*)
END_ACTION
ACTION derevo_write:
_CFC_ (* Continuous Function Chart, elements in execution order *)
_END_CFC_
END_ACTION
ACTION eibPort_climate:
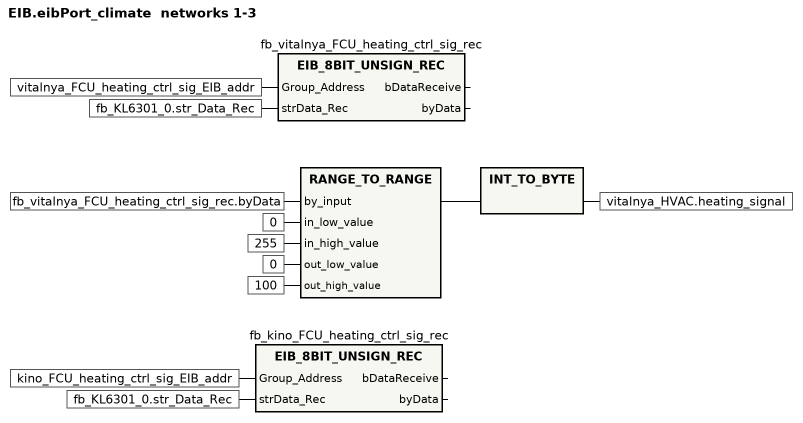
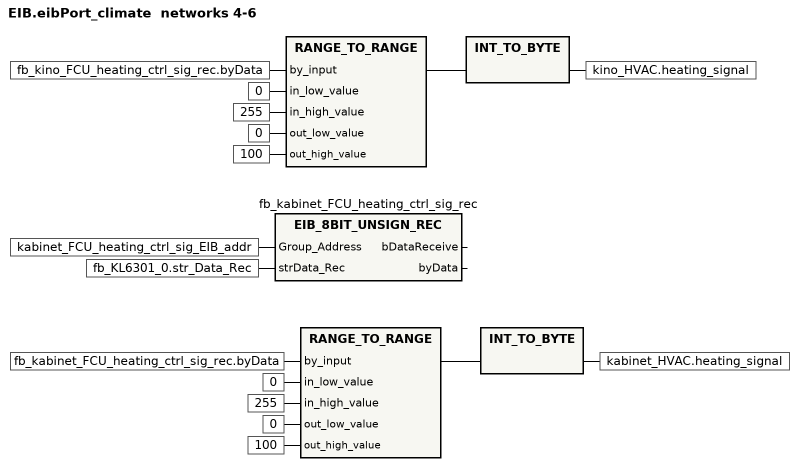
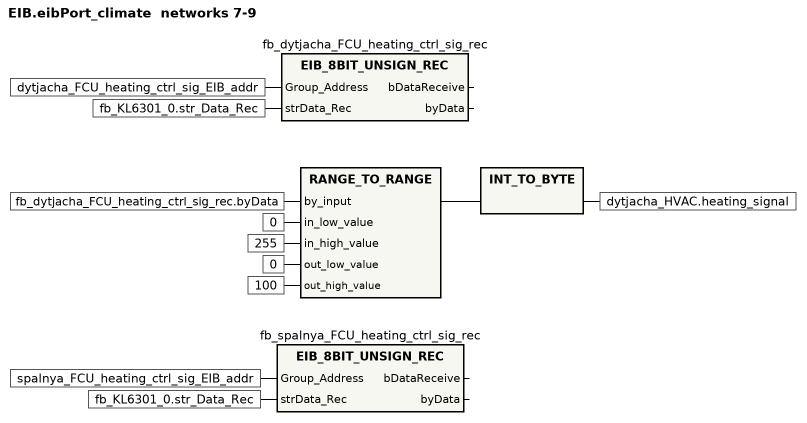
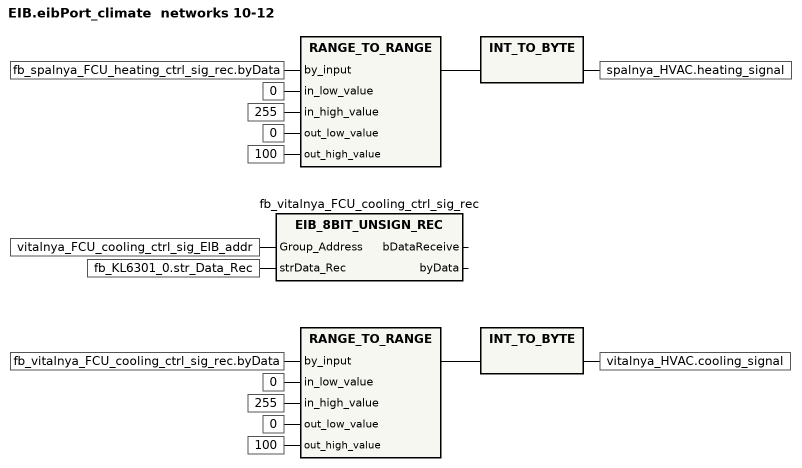
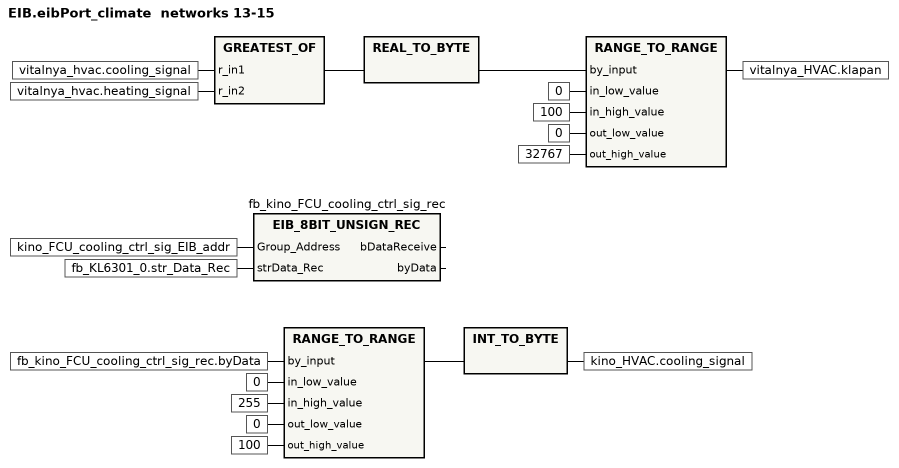
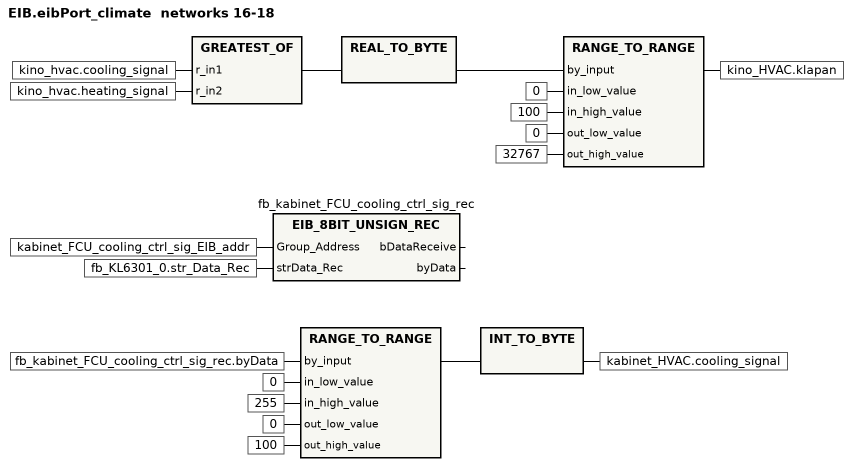
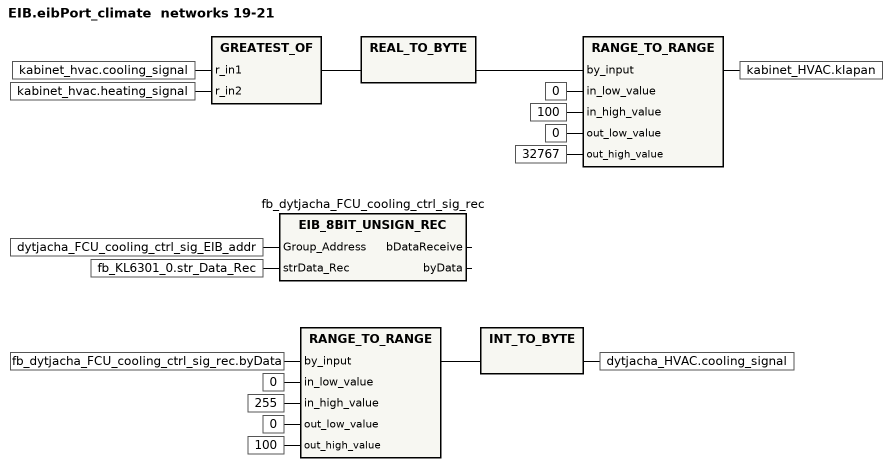
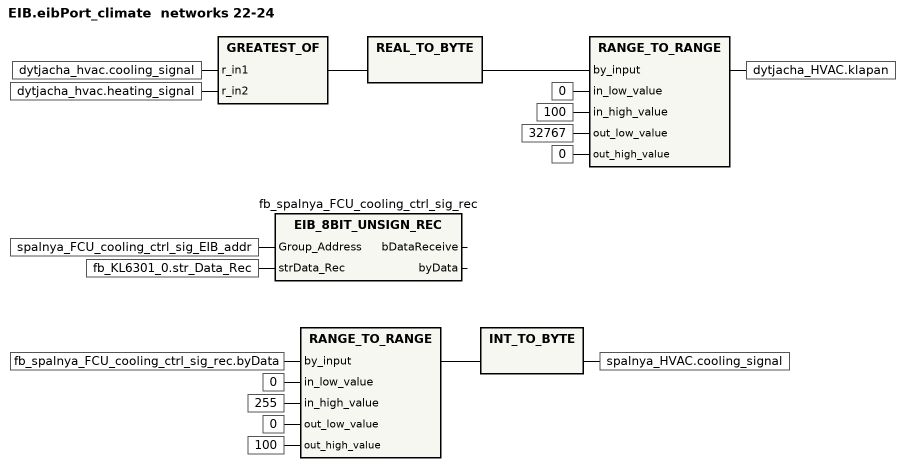
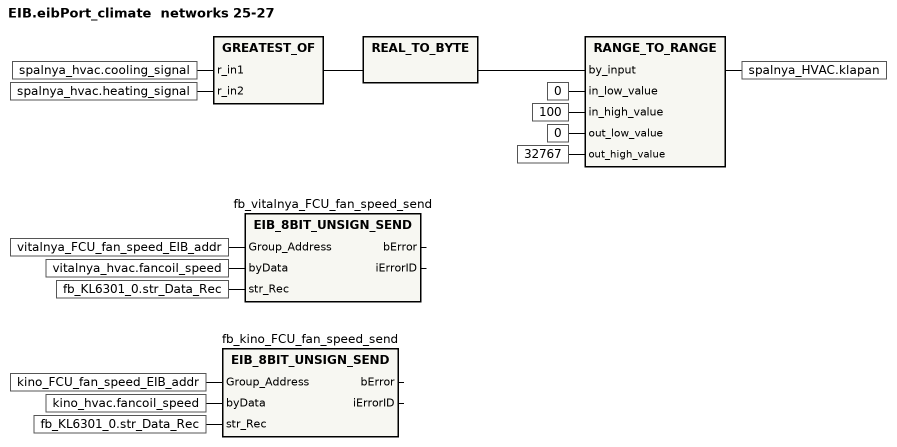
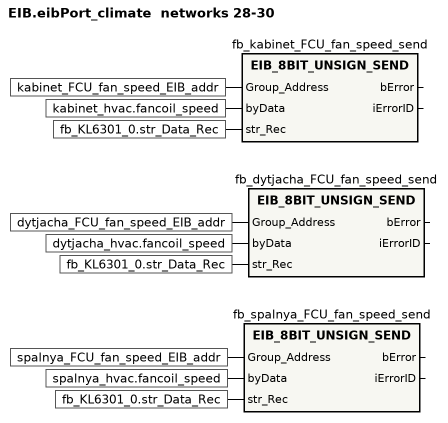
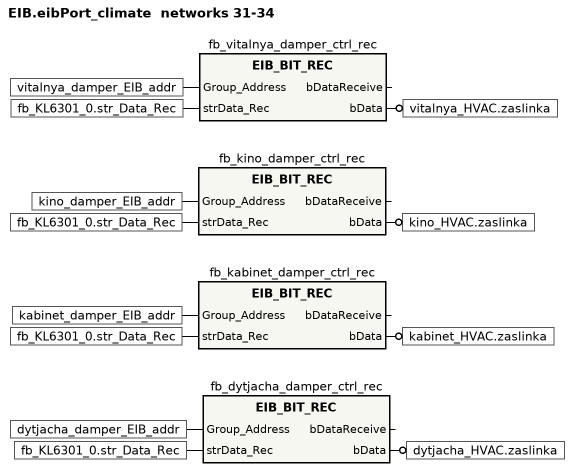
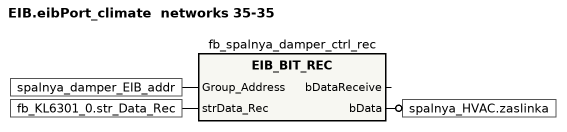
_FBD_ (* Function Block Diagram *)
NETWORK 1
	fb_vitalnya_FCU_heating_ctrl_sig_rec:EIB_8BIT_UNSIGN_REC(Group_Address: vitalnya_FCU_heating_ctrl_sig_EIB_addr, strData_Rec: fb_KL6301_0.str_Data_Rec)
NETWORK 2
	INT_TO_BYTE(RANGE_TO_RANGE(by_input: fb_vitalnya_FCU_heating_ctrl_sig_rec.byData, in_low_value: 0, in_high_value: 255, out_low_value: 0, out_high_value: 100)) => vitalnya_HVAC.heating_signal
NETWORK 3
	fb_kino_FCU_heating_ctrl_sig_rec:EIB_8BIT_UNSIGN_REC(Group_Address: kino_FCU_heating_ctrl_sig_EIB_addr, strData_Rec: fb_KL6301_0.str_Data_Rec)
NETWORK 4
	INT_TO_BYTE(RANGE_TO_RANGE(by_input: fb_kino_FCU_heating_ctrl_sig_rec.byData, in_low_value: 0, in_high_value: 255, out_low_value: 0, out_high_value: 100)) => kino_HVAC.heating_signal
NETWORK 5
	fb_kabinet_FCU_heating_ctrl_sig_rec:EIB_8BIT_UNSIGN_REC(Group_Address: kabinet_FCU_heating_ctrl_sig_EIB_addr, strData_Rec: fb_KL6301_0.str_Data_Rec)
NETWORK 6
	INT_TO_BYTE(RANGE_TO_RANGE(by_input: fb_kabinet_FCU_heating_ctrl_sig_rec.byData, in_low_value: 0, in_high_value: 255, out_low_value: 0, out_high_value: 100)) => kabinet_HVAC.heating_signal
NETWORK 7
	fb_dytjacha_FCU_heating_ctrl_sig_rec:EIB_8BIT_UNSIGN_REC(Group_Address: dytjacha_FCU_heating_ctrl_sig_EIB_addr, strData_Rec: fb_KL6301_0.str_Data_Rec)
NETWORK 8
	INT_TO_BYTE(RANGE_TO_RANGE(by_input: fb_dytjacha_FCU_heating_ctrl_sig_rec.byData, in_low_value: 0, in_high_value: 255, out_low_value: 0, out_high_value: 100)) => dytjacha_HVAC.heating_signal
NETWORK 9
	fb_spalnya_FCU_heating_ctrl_sig_rec:EIB_8BIT_UNSIGN_REC(Group_Address: spalnya_FCU_heating_ctrl_sig_EIB_addr, strData_Rec: fb_KL6301_0.str_Data_Rec)
NETWORK 10
	INT_TO_BYTE(RANGE_TO_RANGE(by_input: fb_spalnya_FCU_heating_ctrl_sig_rec.byData, in_low_value: 0, in_high_value: 255, out_low_value: 0, out_high_value: 100)) => spalnya_HVAC.heating_signal
NETWORK 11
	fb_vitalnya_FCU_cooling_ctrl_sig_rec:EIB_8BIT_UNSIGN_REC(Group_Address: vitalnya_FCU_cooling_ctrl_sig_EIB_addr, strData_Rec: fb_KL6301_0.str_Data_Rec)
NETWORK 12
	INT_TO_BYTE(RANGE_TO_RANGE(by_input: fb_vitalnya_FCU_cooling_ctrl_sig_rec.byData, in_low_value: 0, in_high_value: 255, out_low_value: 0, out_high_value: 100)) => vitalnya_HVAC.cooling_signal
NETWORK 13
	RANGE_TO_RANGE(by_input: REAL_TO_BYTE(GREATEST_OF(r_in1: vitalnya_hvac.cooling_signal, r_in2: vitalnya_hvac.heating_signal)), in_low_value: 0, in_high_value: 100, out_low_value: 0, out_high_value: 32767) => vitalnya_HVAC.klapan
NETWORK 14
	fb_kino_FCU_cooling_ctrl_sig_rec:EIB_8BIT_UNSIGN_REC(Group_Address: kino_FCU_cooling_ctrl_sig_EIB_addr, strData_Rec: fb_KL6301_0.str_Data_Rec)
NETWORK 15
	INT_TO_BYTE(RANGE_TO_RANGE(by_input: fb_kino_FCU_cooling_ctrl_sig_rec.byData, in_low_value: 0, in_high_value: 255, out_low_value: 0, out_high_value: 100)) => kino_HVAC.cooling_signal
NETWORK 16
	RANGE_TO_RANGE(by_input: REAL_TO_BYTE(GREATEST_OF(r_in1: kino_hvac.cooling_signal, r_in2: kino_hvac.heating_signal)), in_low_value: 0, in_high_value: 100, out_low_value: 0, out_high_value: 32767) => kino_HVAC.klapan
NETWORK 17
	fb_kabinet_FCU_cooling_ctrl_sig_rec:EIB_8BIT_UNSIGN_REC(Group_Address: kabinet_FCU_cooling_ctrl_sig_EIB_addr, strData_Rec: fb_KL6301_0.str_Data_Rec)
NETWORK 18
	INT_TO_BYTE(RANGE_TO_RANGE(by_input: fb_kabinet_FCU_cooling_ctrl_sig_rec.byData, in_low_value: 0, in_high_value: 255, out_low_value: 0, out_high_value: 100)) => kabinet_HVAC.cooling_signal
NETWORK 19
	RANGE_TO_RANGE(by_input: REAL_TO_BYTE(GREATEST_OF(r_in1: kabinet_hvac.cooling_signal, r_in2: kabinet_hvac.heating_signal)), in_low_value: 0, in_high_value: 100, out_low_value: 0, out_high_value: 32767) => kabinet_HVAC.klapan
NETWORK 20
	fb_dytjacha_FCU_cooling_ctrl_sig_rec:EIB_8BIT_UNSIGN_REC(Group_Address: dytjacha_FCU_cooling_ctrl_sig_EIB_addr, strData_Rec: fb_KL6301_0.str_Data_Rec)
NETWORK 21
	INT_TO_BYTE(RANGE_TO_RANGE(by_input: fb_dytjacha_FCU_cooling_ctrl_sig_rec.byData, in_low_value: 0, in_high_value: 255, out_low_value: 0, out_high_value: 100)) => dytjacha_HVAC.cooling_signal
NETWORK 22
	RANGE_TO_RANGE(by_input: REAL_TO_BYTE(GREATEST_OF(r_in1: dytjacha_hvac.cooling_signal, r_in2: dytjacha_hvac.heating_signal)), in_low_value: 0, in_high_value: 100, out_low_value: 32767, out_high_value: 0) => dytjacha_HVAC.klapan
NETWORK 23
	fb_spalnya_FCU_cooling_ctrl_sig_rec:EIB_8BIT_UNSIGN_REC(Group_Address: spalnya_FCU_cooling_ctrl_sig_EIB_addr, strData_Rec: fb_KL6301_0.str_Data_Rec)
NETWORK 24
	INT_TO_BYTE(RANGE_TO_RANGE(by_input: fb_spalnya_FCU_cooling_ctrl_sig_rec.byData, in_low_value: 0, in_high_value: 255, out_low_value: 0, out_high_value: 100)) => spalnya_HVAC.cooling_signal
NETWORK 25
	RANGE_TO_RANGE(by_input: REAL_TO_BYTE(GREATEST_OF(r_in1: spalnya_hvac.cooling_signal, r_in2: spalnya_hvac.heating_signal)), in_low_value: 0, in_high_value: 100, out_low_value: 0, out_high_value: 32767) => spalnya_HVAC.klapan
NETWORK 26
	fb_vitalnya_FCU_fan_speed_send:EIB_8BIT_UNSIGN_SEND(Group_Address: vitalnya_FCU_fan_speed_EIB_addr, byData: vitalnya_hvac.fancoil_speed, str_Rec: fb_KL6301_0.str_Data_Rec)
NETWORK 27
	fb_kino_FCU_fan_speed_send:EIB_8BIT_UNSIGN_SEND(Group_Address: kino_FCU_fan_speed_EIB_addr, byData: kino_hvac.fancoil_speed, str_Rec: fb_KL6301_0.str_Data_Rec)
NETWORK 28
	fb_kabinet_FCU_fan_speed_send:EIB_8BIT_UNSIGN_SEND(Group_Address: kabinet_FCU_fan_speed_EIB_addr, byData: kabinet_hvac.fancoil_speed, str_Rec: fb_KL6301_0.str_Data_Rec)
NETWORK 29
	fb_dytjacha_FCU_fan_speed_send:EIB_8BIT_UNSIGN_SEND(Group_Address: dytjacha_FCU_fan_speed_EIB_addr, byData: dytjacha_hvac.fancoil_speed, str_Rec: fb_KL6301_0.str_Data_Rec)
NETWORK 30
	fb_spalnya_FCU_fan_speed_send:EIB_8BIT_UNSIGN_SEND(Group_Address: spalnya_FCU_fan_speed_EIB_addr, byData: spalnya_hvac.fancoil_speed, str_Rec: fb_KL6301_0.str_Data_Rec)
NETWORK 31
	fb_vitalnya_damper_ctrl_rec:EIB_BIT_REC(Group_Address: vitalnya_damper_EIB_addr, strData_Rec: fb_KL6301_0.str_Data_Rec, bData => NOT vitalnya_HVAC.zaslinka)
NETWORK 32
	fb_kino_damper_ctrl_rec:EIB_BIT_REC(Group_Address: kino_damper_EIB_addr, strData_Rec: fb_KL6301_0.str_Data_Rec, bData => NOT kino_HVAC.zaslinka)
NETWORK 33
	fb_kabinet_damper_ctrl_rec:EIB_BIT_REC(Group_Address: kabinet_damper_EIB_addr, strData_Rec: fb_KL6301_0.str_Data_Rec, bData => NOT kabinet_HVAC.zaslinka)
NETWORK 34
	fb_dytjacha_damper_ctrl_rec:EIB_BIT_REC(Group_Address: dytjacha_damper_EIB_addr, strData_Rec: fb_KL6301_0.str_Data_Rec, bData => NOT dytjacha_HVAC.zaslinka)
NETWORK 35
	fb_spalnya_damper_ctrl_rec:EIB_BIT_REC(Group_Address: spalnya_damper_EIB_addr, strData_Rec: fb_KL6301_0.str_Data_Rec, bData => NOT spalnya_HVAC.zaslinka)
_END_FBD_
(* the same logic as Structured Text *)
(* Network 1 *)
fb_vitalnya_FCU_heating_ctrl_sig_rec(Group_Address := vitalnya_FCU_heating_ctrl_sig_EIB_addr, strData_Rec := fb_KL6301_0.str_Data_Rec);
(* Network 2 *)
vitalnya_HVAC.heating_signal := INT_TO_BYTE(RANGE_TO_RANGE(by_input := fb_vitalnya_FCU_heating_ctrl_sig_rec.byData, in_low_value := 0, in_high_value := 255, out_low_value := 0, out_high_value := 100));
(* Network 3 *)
fb_kino_FCU_heating_ctrl_sig_rec(Group_Address := kino_FCU_heating_ctrl_sig_EIB_addr, strData_Rec := fb_KL6301_0.str_Data_Rec);
(* Network 4 *)
kino_HVAC.heating_signal := INT_TO_BYTE(RANGE_TO_RANGE(by_input := fb_kino_FCU_heating_ctrl_sig_rec.byData, in_low_value := 0, in_high_value := 255, out_low_value := 0, out_high_value := 100));
(* Network 5 *)
fb_kabinet_FCU_heating_ctrl_sig_rec(Group_Address := kabinet_FCU_heating_ctrl_sig_EIB_addr, strData_Rec := fb_KL6301_0.str_Data_Rec);
(* Network 6 *)
kabinet_HVAC.heating_signal := INT_TO_BYTE(RANGE_TO_RANGE(by_input := fb_kabinet_FCU_heating_ctrl_sig_rec.byData, in_low_value := 0, in_high_value := 255, out_low_value := 0, out_high_value := 100));
(* Network 7 *)
fb_dytjacha_FCU_heating_ctrl_sig_rec(Group_Address := dytjacha_FCU_heating_ctrl_sig_EIB_addr, strData_Rec := fb_KL6301_0.str_Data_Rec);
(* Network 8 *)
dytjacha_HVAC.heating_signal := INT_TO_BYTE(RANGE_TO_RANGE(by_input := fb_dytjacha_FCU_heating_ctrl_sig_rec.byData, in_low_value := 0, in_high_value := 255, out_low_value := 0, out_high_value := 100));
(* Network 9 *)
fb_spalnya_FCU_heating_ctrl_sig_rec(Group_Address := spalnya_FCU_heating_ctrl_sig_EIB_addr, strData_Rec := fb_KL6301_0.str_Data_Rec);
(* Network 10 *)
spalnya_HVAC.heating_signal := INT_TO_BYTE(RANGE_TO_RANGE(by_input := fb_spalnya_FCU_heating_ctrl_sig_rec.byData, in_low_value := 0, in_high_value := 255, out_low_value := 0, out_high_value := 100));
(* Network 11 *)
fb_vitalnya_FCU_cooling_ctrl_sig_rec(Group_Address := vitalnya_FCU_cooling_ctrl_sig_EIB_addr, strData_Rec := fb_KL6301_0.str_Data_Rec);
(* Network 12 *)
vitalnya_HVAC.cooling_signal := INT_TO_BYTE(RANGE_TO_RANGE(by_input := fb_vitalnya_FCU_cooling_ctrl_sig_rec.byData, in_low_value := 0, in_high_value := 255, out_low_value := 0, out_high_value := 100));
(* Network 13 *)
vitalnya_HVAC.klapan := RANGE_TO_RANGE(by_input := REAL_TO_BYTE(GREATEST_OF(r_in1 := vitalnya_hvac.cooling_signal, r_in2 := vitalnya_hvac.heating_signal)), in_low_value := 0, in_high_value := 100, out_low_value := 0, out_high_value := 32767);
(* Network 14 *)
fb_kino_FCU_cooling_ctrl_sig_rec(Group_Address := kino_FCU_cooling_ctrl_sig_EIB_addr, strData_Rec := fb_KL6301_0.str_Data_Rec);
(* Network 15 *)
kino_HVAC.cooling_signal := INT_TO_BYTE(RANGE_TO_RANGE(by_input := fb_kino_FCU_cooling_ctrl_sig_rec.byData, in_low_value := 0, in_high_value := 255, out_low_value := 0, out_high_value := 100));
(* Network 16 *)
kino_HVAC.klapan := RANGE_TO_RANGE(by_input := REAL_TO_BYTE(GREATEST_OF(r_in1 := kino_hvac.cooling_signal, r_in2 := kino_hvac.heating_signal)), in_low_value := 0, in_high_value := 100, out_low_value := 0, out_high_value := 32767);
(* Network 17 *)
fb_kabinet_FCU_cooling_ctrl_sig_rec(Group_Address := kabinet_FCU_cooling_ctrl_sig_EIB_addr, strData_Rec := fb_KL6301_0.str_Data_Rec);
(* Network 18 *)
kabinet_HVAC.cooling_signal := INT_TO_BYTE(RANGE_TO_RANGE(by_input := fb_kabinet_FCU_cooling_ctrl_sig_rec.byData, in_low_value := 0, in_high_value := 255, out_low_value := 0, out_high_value := 100));
(* Network 19 *)
kabinet_HVAC.klapan := RANGE_TO_RANGE(by_input := REAL_TO_BYTE(GREATEST_OF(r_in1 := kabinet_hvac.cooling_signal, r_in2 := kabinet_hvac.heating_signal)), in_low_value := 0, in_high_value := 100, out_low_value := 0, out_high_value := 32767);
(* Network 20 *)
fb_dytjacha_FCU_cooling_ctrl_sig_rec(Group_Address := dytjacha_FCU_cooling_ctrl_sig_EIB_addr, strData_Rec := fb_KL6301_0.str_Data_Rec);
(* Network 21 *)
dytjacha_HVAC.cooling_signal := INT_TO_BYTE(RANGE_TO_RANGE(by_input := fb_dytjacha_FCU_cooling_ctrl_sig_rec.byData, in_low_value := 0, in_high_value := 255, out_low_value := 0, out_high_value := 100));
(* Network 22 *)
dytjacha_HVAC.klapan := RANGE_TO_RANGE(by_input := REAL_TO_BYTE(GREATEST_OF(r_in1 := dytjacha_hvac.cooling_signal, r_in2 := dytjacha_hvac.heating_signal)), in_low_value := 0, in_high_value := 100, out_low_value := 32767, out_high_value := 0);
(* Network 23 *)
fb_spalnya_FCU_cooling_ctrl_sig_rec(Group_Address := spalnya_FCU_cooling_ctrl_sig_EIB_addr, strData_Rec := fb_KL6301_0.str_Data_Rec);
(* Network 24 *)
spalnya_HVAC.cooling_signal := INT_TO_BYTE(RANGE_TO_RANGE(by_input := fb_spalnya_FCU_cooling_ctrl_sig_rec.byData, in_low_value := 0, in_high_value := 255, out_low_value := 0, out_high_value := 100));
(* Network 25 *)
spalnya_HVAC.klapan := RANGE_TO_RANGE(by_input := REAL_TO_BYTE(GREATEST_OF(r_in1 := spalnya_hvac.cooling_signal, r_in2 := spalnya_hvac.heating_signal)), in_low_value := 0, in_high_value := 100, out_low_value := 0, out_high_value := 32767);
(* Network 26 *)
fb_vitalnya_FCU_fan_speed_send(Group_Address := vitalnya_FCU_fan_speed_EIB_addr, byData := vitalnya_hvac.fancoil_speed, str_Rec := fb_KL6301_0.str_Data_Rec);
(* Network 27 *)
fb_kino_FCU_fan_speed_send(Group_Address := kino_FCU_fan_speed_EIB_addr, byData := kino_hvac.fancoil_speed, str_Rec := fb_KL6301_0.str_Data_Rec);
(* Network 28 *)
fb_kabinet_FCU_fan_speed_send(Group_Address := kabinet_FCU_fan_speed_EIB_addr, byData := kabinet_hvac.fancoil_speed, str_Rec := fb_KL6301_0.str_Data_Rec);
(* Network 29 *)
fb_dytjacha_FCU_fan_speed_send(Group_Address := dytjacha_FCU_fan_speed_EIB_addr, byData := dytjacha_hvac.fancoil_speed, str_Rec := fb_KL6301_0.str_Data_Rec);
(* Network 30 *)
fb_spalnya_FCU_fan_speed_send(Group_Address := spalnya_FCU_fan_speed_EIB_addr, byData := spalnya_hvac.fancoil_speed, str_Rec := fb_KL6301_0.str_Data_Rec);
(* Network 31 *)
fb_vitalnya_damper_ctrl_rec(Group_Address := vitalnya_damper_EIB_addr, strData_Rec := fb_KL6301_0.str_Data_Rec);
vitalnya_HVAC.zaslinka := NOT fb_vitalnya_damper_ctrl_rec.bData;
(* Network 32 *)
fb_kino_damper_ctrl_rec(Group_Address := kino_damper_EIB_addr, strData_Rec := fb_KL6301_0.str_Data_Rec);
kino_HVAC.zaslinka := NOT fb_kino_damper_ctrl_rec.bData;
(* Network 33 *)
fb_kabinet_damper_ctrl_rec(Group_Address := kabinet_damper_EIB_addr, strData_Rec := fb_KL6301_0.str_Data_Rec);
kabinet_HVAC.zaslinka := NOT fb_kabinet_damper_ctrl_rec.bData;
(* Network 34 *)
fb_dytjacha_damper_ctrl_rec(Group_Address := dytjacha_damper_EIB_addr, strData_Rec := fb_KL6301_0.str_Data_Rec);
dytjacha_HVAC.zaslinka := NOT fb_dytjacha_damper_ctrl_rec.bData;
(* Network 35 *)
fb_spalnya_damper_ctrl_rec(Group_Address := spalnya_damper_EIB_addr, strData_Rec := fb_KL6301_0.str_Data_Rec);
spalnya_HVAC.zaslinka := NOT fb_spalnya_damper_ctrl_rec.bData;
END_ACTION
ACTION floor1:
fb_komora_l_read(strData_Rec:=fb_KL6301_0.str_Data_Rec,   Group_Address:=komora_l_adr);
fb_su1_l_read(strData_Rec:=fb_KL6301_0.str_Data_Rec,   Group_Address:=su1_l_adr);
fb_topochna_l_read(strData_Rec:=fb_KL6301_0.str_Data_Rec,  Group_Address:=topochna_l_adr);
fb_su2_bra_read(strData_Rec:=fb_KL6301_0.str_Data_Rec, Group_Address:=su2_bra_adr);
fb_topochna2_l_read(strData_Rec:=fb_KL6301_0.str_Data_Rec, Group_Address:=topochna2_l_adr);
fb_su2_l_read(strData_Rec:=fb_KL6301_0.str_Data_Rec, Group_Address:=su2_l_adr);
fb_su1_rakovyna_read(strData_Rec:=fb_KL6301_0.str_Data_Rec, Group_Address:=su1_rakovyna_adr);
fb_dush_read(strData_Rec:=fb_KL6301_0.str_Data_Rec, Group_Address:=dush_adr);
fb_su2_dush_read(strData_Rec:=fb_KL6301_0.str_Data_Rec, Group_Address:=su2_dush_adr);
fb_vitalnya_smugy2_read(strData_Rec:=fb_KL6301_0.str_Data_Rec, Group_Address:=vitalnya_smugy2_adr);
fb_su2_polytsi_read(strData_Rec:=fb_KL6301_0.str_Data_Rec, Group_Address:=su2_polytsi_adr);
fb_kuhnya1_read(strData_Rec:=fb_KL6301_0.str_Data_Rec, Group_Address:=kuhnya1_adr);
fb_kuhnya2_read(strData_Rec:=fb_KL6301_0.str_Data_Rec, Group_Address:=kuhnya2_adr);
fb_vitalnya_smugy1_read(strData_Rec:=fb_KL6301_0.str_Data_Rec, Group_Address:=vitalnya_smugy1_adr);
fb_vitalnya_l_read(strData_Rec:=fb_KL6301_0.str_Data_Rec, Group_Address:=vitalnya_l_adr);
fb_vitalnya_prokladka_read(strData_Rec:=fb_KL6301_0.str_Data_Rec, Group_Address:=vitalnya_prokladka_adr);
fb_terassa_stina_read(strData_Rec:=fb_KL6301_0.str_Data_Rec, Group_Address:=terassa_stina_adr);
fb_pidval_shody_read(strData_Rec:=fb_KL6301_0.str_Data_Rec, Group_Address:=pidval_shody_adr);
fb_terassa_read(strData_Rec:=fb_KL6301_0.str_Data_Rec, Group_Address:=terassa_adr);
fb_skhody2pov_read(strData_Rec:=fb_KL6301_0.str_Data_Rec, Group_Address:=skhody2pov_adr);
fb_tambur_l_read(strData_Rec:=fb_KL6301_0.str_Data_Rec, Group_Address:=tambur_l_adr);

fb_komora_l_send(str_Rec:=fb_KL6301_0.str_Data_Rec, bData:=komora_l,  Group_Address:=komora_l_adr, bsend:=((fb_komora_l_send.bData XOR fb_komora_l_read.bData XOR komora_l  )OR fb_heartbeat_timer.q))      ;
IF NOT fb_komora_l_read.bDataReceive OR  fb_heartbeat1_timer.q THEN fb_komora_l_send.bSend:=FALSE; fb_komora_l_send(str_Rec:=fb_KL6301_0.str_Data_Rec, bData:=komora_l,  Group_Address:=komora_l_adr);END_IF
fb_su1_l_send(str_Rec:=fb_KL6301_0.str_Data_Rec, bData:=su1_l,  Group_Address:=su1_l_adr, bsend:=(fb_su1_l_read.bData XOR (fb_su1_l_read.bData XOR su1_l)OR fb_heartbeat1_timer.q))      ;
IF NOT fb_su1_l_read.bDataReceive OR  fb_heartbeat1_timer.q THEN fb_su1_l_send.bSend:=FALSE; fb_su1_l_send(str_Rec:=fb_KL6301_0.str_Data_Rec, bData:=su1_l,  Group_Address:=su1_l_adr);END_IF
fb_topochna_l_send(str_Rec:=fb_KL6301_0.str_Data_Rec, bData:=topochna_l,  Group_Address:=topochna_l_adr, bsend:=((fb_topochna_l_send.bData XOR fb_topochna_l_read.bData XOR topochna_l)OR fb_heartbeat1_timer.q))      ;
IF NOT fb_topochna_l_read.bDataReceive OR  fb_heartbeat1_timer.q THEN fb_topochna_l_send.bSend:=FALSE; fb_topochna_l_send(str_Rec:=fb_KL6301_0.str_Data_Rec, bData:=topochna_l,  Group_Address:=topochna_l_adr);END_IF
fb_su2_bra_send(str_Rec:=fb_KL6301_0.str_Data_Rec, bData:=su2_bra,  Group_Address:=su2_bra_adr, bsend:=((fb_su2_bra_read.bData  XOR fb_su2_bra_read.bData XOR su2_bra)OR fb_heartbeat1_timer.q))      ;
IF NOT fb_su2_bra_read.bDataReceive OR  fb_heartbeat1_timer.q THEN fb_su2_bra_send.bSend:=FALSE; fb_su2_bra_send(str_Rec:=fb_KL6301_0.str_Data_Rec, bData:=su2_bra,  Group_Address:=su2_bra_adr);END_IF
fb_topochna2_l_send(str_Rec:=fb_KL6301_0.str_Data_Rec, bData:=topochna2_l,  Group_Address:=topochna2_l_adr, bsend:=((fb_topochna2_l_send.bData XOR fb_topochna2_l_read.bData XOR topochna2_l)OR fb_heartbeat1_timer.q))      ;
IF NOT fb_topochna2_l_read.bDataReceive OR  fb_heartbeat1_timer.q THEN fb_topochna2_l_send.bSend:=FALSE; fb_topochna2_l_send(str_Rec:=fb_KL6301_0.str_Data_Rec, bData:=topochna2_l,  Group_Address:=topochna2_l_adr);END_IF
fb_su2_l_send(str_Rec:=fb_KL6301_0.str_Data_Rec, bData:=su2_l,  Group_Address:=su2_l_adr, bsend:=((fb_su2_l_read.bData  XOR fb_su2_l_read.bData XOR su2_l)OR fb_heartbeat1_timer.q))      ;
IF NOT fb_su2_l_read.bDataReceive OR  fb_heartbeat1_timer.q THEN fb_su2_l_send.bSend:=FALSE; fb_su2_l_send(str_Rec:=fb_KL6301_0.str_Data_Rec, bData:=su2_l,  Group_Address:=su2_l_adr);END_IF
fb_su1_rakovyna_send(str_Rec:=fb_KL6301_0.str_Data_Rec, bData:=su1_rakovyna,  Group_Address:=su1_rakovyna_adr, bsend:=((fb_su1_rakovyna_send.bData XOR fb_su1_rakovyna_read.bData XOR su1_rakovyna)OR fb_heartbeat1_timer.q))      ;
IF NOT fb_su1_rakovyna_read.bDataReceive OR  fb_heartbeat1_timer.q THEN fb_su1_rakovyna_send.bSend:=FALSE; fb_su1_rakovyna_send(str_Rec:=fb_KL6301_0.str_Data_Rec, bData:=su1_rakovyna,  Group_Address:=su1_rakovyna_adr);END_IF
fb_su2_dush_send(str_Rec:=fb_KL6301_0.str_Data_Rec, bData:=su2_dush,  Group_Address:=su2_dush_adr, bsend:=((fb_su2_dush_send.bData XOR fb_su2_dush_read.bData XOR su2_dush)OR fb_heartbeat1_timer.q))      ;
IF NOT fb_su2_dush_read.bDataReceive OR  fb_heartbeat1_timer.q THEN fb_su2_dush_send.bSend:=FALSE; fb_su2_dush_send(str_Rec:=fb_KL6301_0.str_Data_Rec, bData:=su2_dush,  Group_Address:=su2_dush_adr);END_IF
fb_dush_send(str_Rec:=fb_KL6301_0.str_Data_Rec, bData:=dush,  Group_Address:=dush_adr, bsend:=((fb_dush_send.bData XOR fb_dush_read.bData XOR dush)OR fb_heartbeat1_timer.q))      ;
IF NOT fb_dush_read.bDataReceive OR  fb_heartbeat1_timer.q THEN fb_dush_send.bSend:=FALSE; fb_dush_send(str_Rec:=fb_KL6301_0.str_Data_Rec, bData:=dush,  Group_Address:=dush_adr);END_IF
fb_vitalnya_smugy2_send(str_Rec:=fb_KL6301_0.str_Data_Rec, bData:=vitalnya_smugy2,  Group_Address:=vitalnya_smugy2_adr, bsend:=((fb_vitalnya_smugy2_send.bData XOR fb_vitalnya_smugy2_read.bData XOR vitalnya_smugy2)OR fb_heartbeat1_timer.q));   (*       vitalnya_smugy2_read.bData XOR vitalnya_smugy2)) AND fb_heartbeat1_timer.q))      )));*)
IF NOT fb_vitalnya_smugy2_read.bDataReceive OR  fb_heartbeat1_timer.q THEN fb_vitalnya_smugy2_send.bSend:=FALSE; fb_vitalnya_smugy2_send(str_Rec:=fb_KL6301_0.str_Data_Rec, bData:=vitalnya_smugy2,  Group_Address:=vitalnya_smugy2_adr);END_IF
fb_su2_polytsi_send(str_Rec:=fb_KL6301_0.str_Data_Rec, bData:=su2_polytsi,  Group_Address:=su2_polytsi_adr, bsend:=((fb_su2_polytsi_send.bData XOR fb_su2_polytsi_read.bData XOR su2_polytsi)OR fb_heartbeat1_timer.q));   (*       su2_polytsi_read.bData XOR su2_polytsi)) AND fb_heartbeat1_timer.q))      )));*)
IF NOT fb_su2_polytsi_read.bDataReceive OR  fb_heartbeat1_timer.q THEN fb_su2_polytsi_send.bSend:=FALSE; fb_su2_polytsi_send(str_Rec:=fb_KL6301_0.str_Data_Rec, bData:=su2_polytsi,  Group_Address:=su2_polytsi_adr);END_IF
fb_kuhnya1_send(str_Rec:=fb_KL6301_0.str_Data_Rec, bData:=kuhnya1,  Group_Address:=kuhnya1_adr, bsend:=((fb_kuhnya1_send.bData XOR fb_kuhnya1_read.bData XOR kuhnya1)OR fb_heartbeat1_timer.q));   (*       kuhnya1_read.bData XOR kuhnya1)) AND fb_heartbeat1_timer.q))      )));*)
IF NOT fb_kuhnya1_read.bDataReceive OR  fb_heartbeat1_timer.q THEN fb_kuhnya1_send.bSend:=FALSE; fb_kuhnya1_send(str_Rec:=fb_KL6301_0.str_Data_Rec, bData:=kuhnya1,  Group_Address:=kuhnya1_adr);END_IF
fb_kuhnya2_send(str_Rec:=fb_KL6301_0.str_Data_Rec, bData:=kuhnya2,  Group_Address:=kuhnya2_adr, bsend:=((fb_kuhnya2_send.bData XOR fb_kuhnya2_read.bData XOR kuhnya2)OR fb_heartbeat1_timer.q));   (*       kuhnya2_read.bData XOR kuhnya2)) AND fb_heartbeat1_timer.q))      )));*)
IF NOT fb_kuhnya2_read.bDataReceive OR  fb_heartbeat1_timer.q THEN fb_kuhnya2_send.bSend:=FALSE; fb_kuhnya2_send(str_Rec:=fb_KL6301_0.str_Data_Rec, bData:=kuhnya2,  Group_Address:=kuhnya2_adr);END_IF
fb_vitalnya_smugy1_send(str_Rec:=fb_KL6301_0.str_Data_Rec, bData:=vitalnya_smugy1,  Group_Address:=vitalnya_smugy1_adr, bsend:=((fb_vitalnya_smugy1_send.bData XOR fb_vitalnya_smugy1_read.bData XOR vitalnya_smugy1)OR fb_heartbeat1_timer.q));   (*       vitalnya_smugy1_read.bData XOR vitalnya_smugy1)) AND fb_heartbeat1_timer.q))      )));*)
IF NOT fb_vitalnya_smugy1_read.bDataReceive OR  fb_heartbeat1_timer.q THEN fb_vitalnya_smugy1_send.bSend:=FALSE; fb_vitalnya_smugy1_send(str_Rec:=fb_KL6301_0.str_Data_Rec, bData:=vitalnya_smugy1,  Group_Address:=vitalnya_smugy1_adr);END_IF
fb_vitalnya_l_send(str_Rec:=fb_KL6301_0.str_Data_Rec, bData:=vitalnya_l,  Group_Address:=vitalnya_l_adr, bsend:=((fb_vitalnya_l_send.bData XOR fb_vitalnya_l_read.bData XOR vitalnya_l)OR fb_heartbeat1_timer.q));   (*       vitalnya_l_read.bData XOR vitalnya_l)) AND fb_heartbeat1_timer.q))      )));*)
IF NOT fb_vitalnya_l_read.bDataReceive OR  fb_heartbeat1_timer.q THEN fb_vitalnya_l_send.bSend:=FALSE; fb_vitalnya_l_send(str_Rec:=fb_KL6301_0.str_Data_Rec, bData:=vitalnya_l,  Group_Address:=vitalnya_l_adr);END_IF
fb_vitalnya_prokladka_send(str_Rec:=fb_KL6301_0.str_Data_Rec, bData:=vitalnya_prokladka,  Group_Address:=vitalnya_prokladka_adr, bsend:=((fb_vitalnya_prokladka_send.bData XOR fb_vitalnya_prokladka_read.bData XOR vitalnya_prokladka)OR fb_heartbeat1_timer.q));   (*       vitalnya_prokladka_read.bData XOR vitalnya_prokladka)) AND fb_heartbeat1_timer.q))      )));*)
IF NOT fb_vitalnya_prokladka_read.bDataReceive OR  fb_heartbeat1_timer.q THEN fb_vitalnya_prokladka_send.bSend:=FALSE; fb_vitalnya_prokladka_send(str_Rec:=fb_KL6301_0.str_Data_Rec, bData:=vitalnya_prokladka,  Group_Address:=vitalnya_prokladka_adr);END_IF
fb_terassa_stina_send(str_Rec:=fb_KL6301_0.str_Data_Rec, bData:=terassa_stina,  Group_Address:=terassa_stina_adr, bsend:=((fb_terassa_stina_send.bData XOR fb_terassa_stina_read.bData XOR terassa_stina)OR fb_heartbeat1_timer.q));   (*       terassa_stina_read.bData XOR terassa_stina)) AND fb_heartbeat1_timer.q))      )));*)
IF NOT fb_terassa_stina_read.bDataReceive OR  fb_heartbeat1_timer.q THEN fb_terassa_stina_send.bSend:=FALSE; fb_terassa_stina_send(str_Rec:=fb_KL6301_0.str_Data_Rec, bData:=terassa_stina,  Group_Address:=terassa_stina_adr);END_IF
fb_pidval_shody_send(str_Rec:=fb_KL6301_0.str_Data_Rec, bData:=pidval_shody,  Group_Address:=pidval_shody_adr, bsend:=(fb_pidval_shody_read.bData  XOR (fb_pidval_shody_read.bData XOR pidval_shody)OR fb_heartbeat1_timer.q));   (*       pidval_shody_read.bData XOR pidval_shody)) AND fb_heartbeat1_timer.q))      )));*)
IF NOT fb_pidval_shody_read.bDataReceive OR  fb_heartbeat1_timer.q THEN fb_pidval_shody_send.bSend:=FALSE; fb_pidval_shody_send(str_Rec:=fb_KL6301_0.str_Data_Rec, bData:=pidval_shody,  Group_Address:=pidval_shody_adr);END_IF
fb_terassa_send(str_Rec:=fb_KL6301_0.str_Data_Rec, bData:=terassa,  Group_Address:=terassa_adr, bsend:=((fb_terassa_read.bData  XOR fb_terassa_read.bData XOR terassa)OR fb_heartbeat1_timer.q));   (*       terassa_read.bData XOR terassa)) AND fb_heartbeat1_timer.q))      )));*)
IF NOT fb_terassa_read.bDataReceive OR  fb_heartbeat1_timer.q THEN fb_terassa_send.bSend:=FALSE; fb_terassa_send(str_Rec:=fb_KL6301_0.str_Data_Rec, bData:=terassa,  Group_Address:=terassa_adr);END_IF
fb_skhody2pov_send(str_Rec:=fb_KL6301_0.str_Data_Rec, bData:=skhody2pov,  Group_Address:=skhody2pov_adr, bsend:=((fb_skhody2pov_send.bData XOR fb_skhody2pov_read.bData XOR skhody2pov)OR fb_heartbeat1_timer.q));   (*       skhody2pov_read.bData XOR skhody2pov)) AND fb_heartbeat1_timer.q))      )));*)
IF NOT fb_skhody2pov_read.bDataReceive OR  fb_heartbeat1_timer.q THEN fb_skhody2pov_send.bSend:=FALSE; fb_skhody2pov_send(str_Rec:=fb_KL6301_0.str_Data_Rec, bData:=skhody2pov,  Group_Address:=skhody2pov_adr);END_IF
fb_tambur_l_send(str_Rec:=fb_KL6301_0.str_Data_Rec, bData:=tambur_l,  Group_Address:=tambur_l_adr, bsend:=((fb_tambur_l_send.bData XOR fb_tambur_l_read.bData XOR tambur_l)OR fb_heartbeat1_timer.q));   (*       tambur_l_read.bData XOR tambur_l)) AND fb_heartbeat1_timer.q))      )));*)
IF NOT fb_tambur_l_read.bDataReceive OR  fb_heartbeat1_timer.q THEN fb_tambur_l_send.bSend:=FALSE; fb_tambur_l_send(str_Rec:=fb_KL6301_0.str_Data_Rec, bData:=tambur_l,  Group_Address:=tambur_l_adr);END_IF

IF NOT fb_komora_l_read.bDataReceive THEN
	data1floor[100].0:=fb_komora_l_read.bdata;
	komora_l:=fb_komora_l_read.bdata;
ELSE  data1floor[100].0:=komora_l; END_IF;
IF NOT fb_su1_l_read.bDataReceive THEN
	data1floor[100].1:=fb_su1_l_read.bdata;
	su1_l:=fb_su1_l_read.bdata;
ELSE  data1floor[100].1:=su1_l; END_IF;
IF NOT fb_topochna_l_read.bDataReceive THEN
	data1floor[100].2:=fb_topochna_l_read.bdata;
	topochna_l:=fb_topochna_l_read.bdata;
ELSE  data1floor[100].2:=topochna_l; END_IF;
IF NOT fb_su2_bra_read.bDataReceive THEN
	data1floor[100].3:=fb_su2_bra_read.bdata;
	su2_bra:=fb_su2_bra_read.bdata;
ELSE  data1floor[100].3:=su2_bra; END_IF;
IF NOT fb_topochna2_l_read.bDataReceive THEN
	data1floor[100].4:=fb_topochna2_l_read.bdata;
	topochna2_l:=fb_topochna2_l_read.bdata;
ELSE  data1floor[100].4:=topochna2_l; END_IF;
IF NOT fb_su2_l_read.bDataReceive  THEN
	data1floor[100].5:=fb_su2_l_read.bdata;
	su2_l:=fb_su2_l_read.bdata;
ELSE  data1floor[100].5:=su2_l; END_IF;
IF NOT fb_su1_rakovyna_read.bDataReceive THEN
	data1floor[100].6:=fb_su1_rakovyna_read.bdata;
	su1_rakovyna:=fb_su1_rakovyna_read.bdata;
ELSE  data1floor[100].6:=su1_rakovyna; END_IF;
IF NOT fb_su2_dush_read.bDataReceive THEN
	data1floor[100].7:=fb_su2_dush_read.bdata;
	su2_dush:=fb_su2_dush_read.bdata;
ELSE  data1floor[100].7:=su2_dush; END_IF;
IF NOT fb_dush_read.bDataReceive  THEN
	data1floor[101].0:=fb_dush_read.bdata;
	dush:=fb_dush_read.bdata;
ELSE  data1floor[101].0:=dush; END_IF;
IF NOT fb_vitalnya_smugy2_read.bDataReceive THEN
	data1floor[101].1:=fb_vitalnya_smugy2_read.bdata;
	vitalnya_smugy2:=fb_vitalnya_smugy2_read.bdata;
ELSE  data1floor[101].1:=vitalnya_smugy2; END_IF;
IF NOT fb_su2_polytsi_read.bDataReceive  THEN
	data1floor[101].2:=fb_su2_polytsi_read.bdata;
	su2_polytsi:=fb_su2_polytsi_read.bdata;
ELSE  data1floor[101].2:=su2_polytsi; END_IF;
IF NOT fb_kuhnya1_read.bDataReceive  THEN
	data1floor[101].3:=fb_kuhnya1_read.bdata;
	kuhnya1:=fb_kuhnya1_read.bdata;
ELSE  data1floor[101].3:=kuhnya1; END_IF;
IF NOT fb_kuhnya2_read.bDataReceive  THEN
	data1floor[101].4:=fb_kuhnya2_read.bdata;
	kuhnya2:=fb_kuhnya2_read.bdata;
ELSE  data1floor[101].4:=kuhnya2; END_IF;
IF NOT fb_vitalnya_smugy1_read.bDataReceive THEN
	data1floor[101].5:=fb_vitalnya_smugy1_read.bdata;
	vitalnya_smugy1:=fb_vitalnya_smugy1_read.bdata;
ELSE  data1floor[101].5:=vitalnya_smugy1; END_IF;
IF NOT fb_vitalnya_l_read.bDataReceive  THEN
	data1floor[101].6:=fb_vitalnya_l_read.bdata;
	vitalnya_l:=fb_vitalnya_l_read.bdata;
ELSE  data1floor[101].6:=vitalnya_l; END_IF;
IF NOT fb_vitalnya_prokladka_read.bDataReceive  THEN
	data1floor[101].7:=fb_vitalnya_prokladka_read.bdata;
	vitalnya_prokladka:=fb_vitalnya_prokladka_read.bdata;
ELSE  data1floor[101].7:=vitalnya_prokladka; END_IF;
IF NOT fb_terassa_stina_read.bDataReceive THEN
	data1floor[102].0:=fb_terassa_stina_read.bdata;
	terassa_stina:=fb_terassa_stina_read.bdata;
 ELSE  data1floor[102].0:=terassa_stina; END_IF;
IF NOT fb_pidval_shody_read.bDataReceive  THEN
	data1floor[102].1:=fb_pidval_shody_read.bdata;
	pidval_shody:=fb_pidval_shody_read.bdata;
ELSE  data1floor[102].1:=pidval_shody; END_IF;
IF NOT fb_terassa_read.bDataReceive  THEN
	data1floor[102].2:=fb_terassa_read.bdata;
	terassa:=fb_terassa_read.bdata;
ELSE data1floor[102].2:=terassa; END_IF;
IF NOT fb_skhody2pov_read.bDataReceive THEN
	data1floor[102].3:=fb_skhody2pov_read.bdata;
	skhody2pov:=fb_skhody2pov_read.bdata;
 ELSE  data1floor[102].3:=skhody2pov; END_IF;
IF NOT fb_tambur_l_read.bDataReceive  THEN
	data1floor[102].4:=fb_tambur_l_read.bdata;
	tambur_l:=fb_tambur_l_read.bdata;
ELSE  data1floor[102].4:=tambur_l; END_IF;
END_ACTION
ACTION floor2:
fb_balkon_peryla_read(strData_Rec:=fb_KL6301_0.str_Data_Rec, Group_Address:=balkon_peryla_adr);
fb_kino_l_read(strData_Rec:=fb_KL6301_0.str_Data_Rec, Group_Address:=kino_l_adr);
fb_balkon_bra_read(strData_Rec:=fb_KL6301_0.str_Data_Rec, Group_Address:=balkon_bra_adr);
fb_kabinet_balkon_l_read(strData_Rec:=fb_KL6301_0.str_Data_Rec, Group_Address:=kabinet_balkon_l_adr);
fb_balkon_read(strData_Rec:=fb_KL6301_0.str_Data_Rec, Group_Address:=balkon_adr);
fb_korydor1_read(strData_Rec:=fb_KL6301_0.str_Data_Rec, Group_Address:=korydor1_adr);
fb_kino_bra_read(strData_Rec:=fb_KL6301_0.str_Data_Rec, Group_Address:=kino_bra_adr);
fb_korydor2_read(strData_Rec:=fb_KL6301_0.str_Data_Rec,  Group_Address:=korydor2_adr);
fb_studio_pidsvitka_read(strData_Rec:=fb_KL6301_0.str_Data_Rec, Group_Address:=studio_pidsvitka_adr);
fb_skhody2_3_read(strData_Rec:=fb_KL6301_0.str_Data_Rec, Group_Address:=skhody2_3_adr);
fb_studio_l_read(strData_Rec:=fb_KL6301_0.str_Data_Rec, Group_Address:=studio_l_adr);
fb_kabinet_pidsvitka_kolo_read(strData_Rec:=fb_KL6301_0.str_Data_Rec, Group_Address:=kabinet_pidsvitka_kolo_adr);
fb_kabinet_svitlo_read(strData_Rec:=fb_KL6301_0.str_Data_Rec, Group_Address:=kabinet_svitlo_adr);
fb_stend_read(strData_Rec:=fb_KL6301_0.str_Data_Rec, Group_Address:=stend_adr);
fb_kabinet_kobra_read(strData_Rec:=fb_KL6301_0.str_Data_Rec, Group_Address:=kabinet_kobra_adr);
fb_skhody_peryla_read(strData_Rec:=fb_KL6301_0.str_Data_Rec,Group_Address:=skhody_peryla_adr);
fb_tambur2_read(strData_Rec:=fb_KL6301_0.str_Data_Rec, Group_Address:=tambur2_adr);

fb_balkon_peryla_send(str_Rec:=fb_KL6301_0.str_Data_Rec, bData:=balkon_peryla,  Group_Address:=balkon_peryla_adr, bsend:=((fb_balkon_peryla_send.bData XOR fb_balkon_peryla_read.bData XOR balkon_peryla)OR fb_heartbeat2_timer.q));   (*       balkon_peryla_read.bData XOR balkon_peryla)) AND fb_heartbeat2_timer.q))      )));*)
IF NOT fb_balkon_peryla_read.bDataReceive OR  fb_heartbeat2_timer.q THEN fb_balkon_peryla_send.bSend:=FALSE; fb_balkon_peryla_send(str_Rec:=fb_KL6301_0.str_Data_Rec, bData:=balkon_peryla,  Group_Address:=balkon_peryla_adr);END_IF
fb_kino_l_send(str_Rec:=fb_KL6301_0.str_Data_Rec, bData:=kino_l,  Group_Address:=kino_l_adr, bsend:=((fb_kino_l_send.bData  <>  fb_kino_l_read.bData <> kino_l)OR fb_heartbeat2_timer.q));
IF NOT fb_kino_l_read.bDataReceive OR  fb_heartbeat2_timer.q THEN fb_kino_l_send.bSend:=FALSE; fb_kino_l_send(str_Rec:=fb_KL6301_0.str_Data_Rec,  Group_Address:=kino_l_adr);END_IF
fb_balkon_bra_send(str_Rec:=fb_KL6301_0.str_Data_Rec, bData:=balkon_bra,  Group_Address:=balkon_bra_adr, bsend:=((fb_balkon_bra_read.bData  XOR fb_balkon_bra_read.bData XOR balkon_bra)OR fb_heartbeat2_timer.q));   (*       balkon_bra_read.bData XOR balkon_bra)) AND fb_heartbeat2_timer.q))      )));*)
IF NOT fb_balkon_bra_read.bDataReceive OR  fb_heartbeat2_timer.q THEN fb_balkon_bra_send.bSend:=FALSE; fb_balkon_bra_send(str_Rec:=fb_KL6301_0.str_Data_Rec, bData:=balkon_bra,  Group_Address:=balkon_bra_adr);END_IF
fb_kabinet_balkon_l_send(str_Rec:=fb_KL6301_0.str_Data_Rec, bData:=kabinet_balkon_l,  Group_Address:=kabinet_balkon_l_adr, bsend:=(( fb_kabinet_balkon_l_send.bData XOR fb_kabinet_balkon_l_read.bData XOR kabinet_balkon_l)OR fb_heartbeat2_timer.q));   (*       kabinet_balkon_l_read.bData XOR kabinet_balkon_l)) AND fb_heartbeat2_timer.q))      )));*)
IF NOT fb_kabinet_balkon_l_read.bDataReceive OR  fb_heartbeat2_timer.q THEN fb_kabinet_balkon_l_send.bSend:=FALSE; fb_kabinet_balkon_l_send(str_Rec:=fb_KL6301_0.str_Data_Rec, bData:=kabinet_balkon_l,  Group_Address:=kabinet_balkon_l_adr);END_IF
fb_balkon_send(str_Rec:=fb_KL6301_0.str_Data_Rec, bData:=balkon,  Group_Address:=balkon_adr, bsend:=((fb_balkon_send.bData XOR fb_balkon_read.bData XOR balkon)OR fb_heartbeat2_timer.q));   (*       balkon_read.bData XOR balkon)) AND fb_heartbeat2_timer.q))      )));*)
IF NOT fb_balkon_read.bDataReceive OR  fb_heartbeat2_timer.q THEN fb_balkon_send.bSend:=FALSE; fb_balkon_send(str_Rec:=fb_KL6301_0.str_Data_Rec, bData:=balkon,  Group_Address:=balkon_adr);END_IF
fb_korydor1_send(str_Rec:=fb_KL6301_0.str_Data_Rec, bData:=korydor1,  Group_Address:=korydor1_adr, bsend:=((fb_korydor1_send.bData XOR fb_korydor1_read.bData XOR korydor1)OR fb_heartbeat2_timer.q));   (* *)
IF NOT fb_korydor1_read.bDataReceive OR  fb_heartbeat2_timer.q THEN fb_korydor1_send.bSend:=FALSE; fb_korydor1_send(str_Rec:=fb_KL6301_0.str_Data_Rec, bData:=korydor1,  Group_Address:=korydor1_adr);END_IF
fb_kino_bra_send(str_Rec:=fb_KL6301_0.str_Data_Rec, bData:=kino_bra,  Group_Address:=kino_bra_adr, bsend:=((fb_kino_bra_send.bData XOR fb_kino_bra_read.bData XOR kino_bra)OR fb_heartbeat2_timer.q));
IF NOT fb_kino_bra_read.bDataReceive OR  fb_heartbeat2_timer.q THEN fb_kino_bra_send.bSend:=FALSE; fb_kino_bra_send(str_Rec:=fb_KL6301_0.str_Data_Rec, bData:=kino_bra,  Group_Address:=kino_bra_adr);END_IF
fb_korydor2_send(str_Rec:=fb_KL6301_0.str_Data_Rec, bData:=korydor2,  Group_Address:=korydor2_adr, bsend:=((fb_korydor2_send.bData XOR fb_korydor2_read.bData XOR korydor2)OR fb_heartbeat2_timer.q));
IF NOT fb_korydor2_read.bDataReceive OR  fb_heartbeat2_timer.q THEN fb_korydor2_send.bSend:=FALSE; fb_korydor2_send(str_Rec:=fb_KL6301_0.str_Data_Rec, bData:=korydor2,  Group_Address:=korydor2_adr);END_IF
fb_studio_pidsvitka_send(str_Rec:=fb_KL6301_0.str_Data_Rec, bData:=studio_pidsvitka,  Group_Address:=studio_pidsvitka_adr, bsend:=((fb_studio_pidsvitka_send.bData XOR fb_studio_pidsvitka_read.bData XOR studio_pidsvitka)OR fb_heartbeat2_timer.q));
IF NOT fb_studio_pidsvitka_read.bDataReceive OR  fb_heartbeat2_timer.q THEN fb_studio_pidsvitka_send.bSend:=FALSE; fb_studio_pidsvitka_send(str_Rec:=fb_KL6301_0.str_Data_Rec, bData:=studio_pidsvitka,  Group_Address:=studio_pidsvitka_adr);END_IF
fb_skhody2_3_send(str_Rec:=fb_KL6301_0.str_Data_Rec, bData:=skhody2_3,  Group_Address:=skhody2_3_adr, bsend:=((fb_skhody2_3_send.bData XOR fb_skhody2_3_read.bData XOR skhody2_3)OR fb_heartbeat2_timer.q));
IF NOT fb_skhody2_3_read.bDataReceive OR  fb_heartbeat2_timer.q THEN fb_skhody2_3_send.bSend:=FALSE; fb_skhody2_3_send(str_Rec:=fb_KL6301_0.str_Data_Rec, bData:=skhody2_3,  Group_Address:=skhody2_3_adr);END_IF
fb_studio_l_send(str_Rec:=fb_KL6301_0.str_Data_Rec, bData:=studio_l,  Group_Address:=studio_l_adr, bsend:=((fb_studio_l_send.bData XOR fb_studio_l_read.bData XOR studio_l)OR fb_heartbeat2_timer.q));
IF NOT fb_studio_l_read.bDataReceive OR  fb_heartbeat2_timer.q THEN fb_studio_l_send.bSend:=FALSE; fb_studio_l_send(str_Rec:=fb_KL6301_0.str_Data_Rec, bData:=studio_l,  Group_Address:=studio_l_adr);END_IF
fb_kabinet_pidsvitka_kolo_send(str_Rec:=fb_KL6301_0.str_Data_Rec, bData:=kabinet_pidsvitka_kolo,  Group_Address:=kabinet_pidsvitka_kolo_adr, bsend:=((fb_kabinet_pidsvitka_kolo_send.bData XOR fb_kabinet_pidsvitka_kolo_read.bData XOR kabinet_pidsvitka_kolo)OR fb_heartbeat2_timer.q));
IF NOT fb_kabinet_pidsvitka_kolo_read.bDataReceive OR  fb_heartbeat2_timer.q THEN fb_kabinet_pidsvitka_kolo_send.bSend:=FALSE; fb_kabinet_pidsvitka_kolo_send(str_Rec:=fb_KL6301_0.str_Data_Rec, bData:=kabinet_pidsvitka_kolo,  Group_Address:=kabinet_pidsvitka_kolo_adr);END_IF
fb_kabinet_svitlo_send(str_Rec:=fb_KL6301_0.str_Data_Rec, bData:=kabinet_svitlo,  Group_Address:=kabinet_svitlo_adr, bsend:=((fb_kabinet_svitlo_send.bData XOR fb_kabinet_svitlo_read.bData XOR kabinet_svitlo)OR fb_heartbeat2_timer.q));
IF NOT fb_kabinet_svitlo_read.bDataReceive OR  fb_heartbeat2_timer.q THEN fb_kabinet_svitlo_send.bSend:=FALSE; fb_kabinet_svitlo_send(str_Rec:=fb_KL6301_0.str_Data_Rec, bData:=kabinet_svitlo,  Group_Address:=kabinet_svitlo_adr);END_IF
fb_stend_send(str_Rec:=fb_KL6301_0.str_Data_Rec, bData:=stend,  Group_Address:=stend_adr, bsend:=((fb_stend_send.bData XOR fb_stend_read.bData XOR stend)OR fb_heartbeat2_timer.q));
IF NOT fb_stend_read.bDataReceive OR  fb_heartbeat2_timer.q THEN fb_stend_send.bSend:=FALSE; fb_stend_send(str_Rec:=fb_KL6301_0.str_Data_Rec, bData:=stend,  Group_Address:=stend_adr);END_IF
fb_kabinet_kobra_send(str_Rec:=fb_KL6301_0.str_Data_Rec, bData:=kabinet_kobra,  Group_Address:=kabinet_kobra_adr, bsend:=((fb_kabinet_kobra_send.bData XOR fb_kabinet_kobra_read.bData XOR kabinet_kobra)OR fb_heartbeat2_timer.q));
IF NOT fb_kabinet_kobra_read.bDataReceive OR  fb_heartbeat2_timer.q THEN fb_kabinet_kobra_send.bSend:=FALSE; fb_kabinet_kobra_send(str_Rec:=fb_KL6301_0.str_Data_Rec, bData:=kabinet_kobra,  Group_Address:=kabinet_kobra_adr);END_IF
fb_skhody_peryla_send(str_Rec:=fb_KL6301_0.str_Data_Rec, bData:=skhody_peryla,  Group_Address:=skhody_peryla_adr, bsend:=((fb_skhody_peryla_send.bData XOR fb_skhody_peryla_read.bData XOR skhody_peryla)OR fb_heartbeat2_timer.q));
IF NOT fb_skhody_peryla_read.bDataReceive OR  fb_heartbeat2_timer.q THEN fb_skhody_peryla_send.bSend:=FALSE; fb_skhody_peryla_send(str_Rec:=fb_KL6301_0.str_Data_Rec, bData:=skhody_peryla,  Group_Address:=skhody_peryla_adr);END_IF
fb_tambur2_send(str_Rec:=fb_KL6301_0.str_Data_Rec, bData:=tambur2,  Group_Address:=tambur2_adr, bsend:=((fb_tambur2_send.bData XOR fb_tambur2_read.bData XOR tambur2)OR fb_heartbeat2_timer.q)) ;
IF NOT fb_tambur2_read.bDataReceive OR  fb_heartbeat2_timer.q THEN fb_tambur2_send.bSend:=FALSE; fb_tambur2_send(str_Rec:=fb_KL6301_0.str_Data_Rec, bData:=tambur2,  Group_Address:=tambur2_adr);END_IF

IF NOT  fb_balkon_peryla_read.bDataReceive THEN
	data2floor[100].0:=fb_balkon_peryla_read.bdata;
	balkon_peryla:=fb_balkon_peryla_read.bdata;
ELSE data2floor[100].0:=balkon_peryla; END_IF
IF NOT fb_kino_l_read.bDataReceive THEN
	data2floor[100].1:=fb_kino_l_read.bdata;
	kino_l:=fb_kino_l_read.bdata;
ELSE data2floor[100].1:=kino_l; END_IF
IF NOT fb_balkon_bra_read.bDataReceive THEN
	data2floor[100].2:= fb_balkon_bra_read.bdata;
	balkon_bra:= fb_balkon_bra_read.bdata;
ELSE data2floor[100].2:= balkon_bra;END_IF
IF NOT fb_kabinet_balkon_l_read.bDataReceive  THEN
	 data2floor[100].3:=fb_kabinet_balkon_l_read.bdata;
	kabinet_balkon_l:=fb_kabinet_balkon_l_read.bdata;
ELSE 	data2floor[100].3:=kabinet_balkon_l; END_IF
IF NOT fb_balkon_read.bDataReceive THEN
	data2floor[100].4:=fb_balkon_read.bdata;
	balkon:=fb_balkon_read.bdata;
ELSE 	data2floor[100].4:=balkon; END_IF
IF NOT fb_korydor1_read.bDataReceive THEN
	data2floor[100].5:=fb_korydor1_read.bdata;
	korydor1:=fb_korydor1_read.bdata;
ELSE 	data2floor[100].5:=korydor1;END_IF;
IF NOT fb_kino_bra_read.bDataReceive  THEN
	data2floor[100].6:=fb_kino_bra_read.bdata;
	kino_bra:=fb_kino_bra_read.bdata;
 ELSE 	data2floor[100].6:=kino_bra; END_IF;
IF NOT fb_korydor2_read.bDataReceive  THEN
	data2floor[100].7:=fb_korydor2_read.bdata;
	korydor2:=fb_korydor2_read.bdata;
ELSE 	data2floor[100].7:=korydor2; END_IF;
IF NOT fb_studio_pidsvitka_read.bDataReceive  THEN
	data2floor[101].0:=fb_studio_pidsvitka_read.bdata;
	studio_pidsvitka:=fb_studio_pidsvitka_read.bdata;
ELSE data2floor[101].0:=studio_pidsvitka; END_IF;
IF NOT fb_skhody2_3_read.bDataReceive  THEN
	data2floor[101].1:=fb_skhody2_3_read.bdata;
	skhody2_3:=fb_skhody2_3_read.bdata;
ELSE data2floor[101].1:=skhody2_3; END_IF;
IF NOT fb_studio_l_read.bDataReceive THEN
	data2floor[101].2:=fb_studio_l_read.bdata;
	studio_l:=fb_studio_l_read.bdata;
ELSE data2floor[101].2:=studio_l; END_IF;
IF NOT fb_kabinet_pidsvitka_kolo_read.bDataReceive THEN
	data2floor[101].3:=fb_kabinet_pidsvitka_kolo_read.bdata;
	kabinet_pidsvitka_kolo:=fb_kabinet_pidsvitka_kolo_read.bdata;
ELSE data2floor[101].3:=kabinet_pidsvitka_kolo; END_IF;
IF NOT fb_kabinet_svitlo_read.bDataReceive THEN
	data2floor[101].4:=fb_kabinet_svitlo_read.bdata;
	kabinet_svitlo:=fb_kabinet_svitlo_read.bdata;
ELSE data2floor[101].4:=kabinet_svitlo; END_IF;
IF NOT fb_kabinet_kobra_read.bDataReceive THEN
	data2floor[101].5:=fb_kabinet_kobra_read.bdata;
	kabinet_kobra:=fb_kabinet_kobra_read.bdata;
ELSE data2floor[101].5:=kabinet_kobra; END_IF;
IF NOT fb_tambur2_read.bDataReceive  THEN
	data2floor[101].6:=fb_tambur2_read.bdata;
	tambur2:=fb_tambur2_read.bdata;
ELSE data2floor[101].6:=tambur2; END_IF;
IF NOT fb_stend_read.bDataReceive  THEN
	data2floor[101].7:=fb_stend_read.bdata;
	stend:=fb_stend_read.bdata;
ELSE  data2floor[101].7:=stend; END_IF;
IF NOT fb_skhody_peryla_read.bDataReceive  THEN
	data2floor[102].0:=fb_skhody_peryla_read.bdata;
	skhody_peryla:=fb_skhody_peryla_read.bdata;
ELSE data2floor[102].0:=skhody_peryla; END_IF;
END_ACTION
ACTION floor3:
(*read*)
fb_spalnya_kontrazhur_read(strData_Rec:=fb_KL6301_0.str_Data_Rec, Group_Address:=spalnya_kontrazhur_adr);
fb_spalnya_balkon_read(strData_Rec:=fb_KL6301_0.str_Data_Rec,  Group_Address:=spalnya_balkon_adr);
fb_spalnya_kulbaba_read(strData_Rec:=fb_KL6301_0.str_Data_Rec, Group_Address:=spalnya_kulbaba_adr);
fb_spalnya_kontrazhur_b_read(strData_Rec:=fb_KL6301_0.str_Data_Rec, Group_Address:=spalnya_kontrazhur_b_adr);
fb_spalnya_kontrazhur_l_read(strData_Rec:=fb_KL6301_0.str_Data_Rec, Group_Address:=spalnya_kontrazhur_l_adr);
fb_su3_stina_read(strData_Rec:=fb_KL6301_0.str_Data_Rec, Group_Address:=su3_stina_adr);
fb_su3_pidsvitka_read(strData_Rec:=fb_KL6301_0.str_Data_Rec,  Group_Address:=su3_pidsvitka_adr);
fb_su3_bra_read(strData_Rec:=fb_KL6301_0.str_Data_Rec, Group_Address:=su3_bra_adr);
fb_su3_kontrazhur_read(strData_Rec:=fb_KL6301_0.str_Data_Rec, Group_Address:=su3_kontrazhur_adr);
fb_su3_kontrazhur_k_read(strData_Rec:=fb_KL6301_0.str_Data_Rec,  Group_Address:=su3_kontrazhur_k_adr);
fb_su3_lampa_read(strData_Rec:=fb_KL6301_0.str_Data_Rec, Group_Address:=su3_lampa_adr);
fb_dytjacha_read(strData_Rec:=fb_KL6301_0.str_Data_Rec, Group_Address:=dytjacha_adr);
fb_dytjacha_bra_read(strData_Rec:=fb_KL6301_0.str_Data_Rec, Group_Address:=dytjacha_bra_adr);
fb_garderob_read(strData_Rec:=fb_KL6301_0.str_Data_Rec, Group_Address:=garderob_adr);
fb_bar_read(strData_Rec:=fb_KL6301_0.str_Data_Rec, Group_Address:=bar_adr);
fb_korydor_skeli_read(strData_Rec:=fb_KL6301_0.str_Data_Rec, Group_Address:=korydor_skeli_adr);
fb_choven_read(strData_Rec:=fb_KL6301_0.str_Data_Rec, Group_Address:=choven_adr);
fb_korydor_lampa_read(strData_Rec:=fb_KL6301_0.str_Data_Rec, Group_Address:=korydor_lampa_adr);
fb_serverna_read(strData_Rec:=fb_KL6301_0.str_Data_Rec, Group_Address:=serverna_adr);
fb_korydor_svitlo_read(strData_Rec:=fb_KL6301_0.str_Data_Rec, Group_Address:=korydor_svitlo_adr);
fb_moove_sensors_read(strData_Rec:=fb_KL6301_0.str_Data_Rec, Group_Address:=moove_sensors_adr);

fb_spalnya_kontrazhur_send(str_Rec:=fb_KL6301_0.str_Data_Rec, bData:=spalnya_kontrazhur,  Group_Address:=spalnya_kontrazhur_adr, bsend:=((fb_spalnya_kontrazhur_send.bData XOR fb_spalnya_kontrazhur_read.bData XOR spalnya_kontrazhur)OR fb_heartbeat_timer.q));
IF NOT fb_spalnya_kontrazhur_read.bDataReceive OR  fb_heartbeat_timer.q THEN fb_spalnya_kontrazhur_send.bSend:=FALSE; fb_spalnya_kontrazhur_send(str_Rec:=fb_KL6301_0.str_Data_Rec, bData:=spalnya_kontrazhur,  Group_Address:=spalnya_kontrazhur_adr);END_IF
fb_spalnya_balkon_send(str_Rec:=fb_KL6301_0.str_Data_Rec, bData:=spalnya_balkon,  Group_Address:=spalnya_balkon_adr, bsend:=((fb_spalnya_balkon_send.bData XOR fb_spalnya_balkon_read.bData XOR spalnya_balkon)OR fb_heartbeat_timer.q));
IF NOT fb_spalnya_balkon_read.bDataReceive OR  fb_heartbeat_timer.q THEN fb_spalnya_balkon_send.bSend:=FALSE; fb_spalnya_balkon_send(str_Rec:=fb_KL6301_0.str_Data_Rec, bData:=spalnya_balkon,  Group_Address:=spalnya_balkon_adr);END_IF
fb_spalnya_kulbaba_send(str_Rec:=fb_KL6301_0.str_Data_Rec, bData:=spalnya_kulbaba,  Group_Address:=spalnya_kulbaba_adr, bsend:=((fb_spalnya_kulbaba_send.bData XOR fb_spalnya_kulbaba_read.bData XOR spalnya_kulbaba)OR fb_heartbeat_timer.q));
IF NOT fb_spalnya_kulbaba_read.bDataReceive OR  fb_heartbeat_timer.q THEN fb_spalnya_kulbaba_send.bSend:=FALSE; fb_spalnya_kulbaba_send(str_Rec:=fb_KL6301_0.str_Data_Rec, bData:=spalnya_kulbaba,  Group_Address:=spalnya_kulbaba_adr);END_IF
fb_spalnya_kontrazhur_b_send(str_Rec:=fb_KL6301_0.str_Data_Rec, bData:=spalnya_kontrazhur_b,  Group_Address:=spalnya_kontrazhur_b_adr, bsend:=((fb_spalnya_kontrazhur_b_send.bData XOR fb_spalnya_kontrazhur_b_read.bData XOR spalnya_kontrazhur_b)OR fb_heartbeat_timer.q));
IF NOT fb_spalnya_kontrazhur_b_read.bDataReceive OR  fb_heartbeat_timer.q THEN fb_spalnya_kontrazhur_b_send.bSend:=FALSE; fb_spalnya_kontrazhur_b_send(str_Rec:=fb_KL6301_0.str_Data_Rec, bData:=spalnya_kontrazhur_b,  Group_Address:=spalnya_kontrazhur_b_adr);END_IF
fb_spalnya_kontrazhur_l_send(str_Rec:=fb_KL6301_0.str_Data_Rec, bData:=spalnya_kontrazhur_l,  Group_Address:=spalnya_kontrazhur_l_adr, bsend:=((fb_spalnya_kontrazhur_l_send.bData XOR fb_spalnya_kontrazhur_l_read.bData XOR spalnya_kontrazhur_l)OR fb_heartbeat_timer.q));
IF NOT fb_spalnya_kontrazhur_l_read.bDataReceive OR  fb_heartbeat_timer.q THEN fb_spalnya_kontrazhur_l_send.bSend:=FALSE; fb_spalnya_kontrazhur_l_send(str_Rec:=fb_KL6301_0.str_Data_Rec, bData:=spalnya_kontrazhur_l,  Group_Address:=spalnya_kontrazhur_l_adr);END_IF
fb_su3_stina_send(str_Rec:=fb_KL6301_0.str_Data_Rec, bData:=su3_stina,  Group_Address:=su3_stina_adr, bsend:=((fb_su3_stina_send.bData XOR fb_su3_stina_read.bData XOR su3_stina)OR fb_heartbeat_timer.q));
IF NOT fb_su3_stina_read.bDataReceive OR  fb_heartbeat_timer.q THEN fb_su3_stina_send.bSend:=FALSE; fb_su3_stina_send(str_Rec:=fb_KL6301_0.str_Data_Rec, bData:=su3_stina,  Group_Address:=su3_stina_adr);END_IF
fb_su3_pidsvitka_send(str_Rec:=fb_KL6301_0.str_Data_Rec, bData:=su3_pidsvitka,  Group_Address:=su3_pidsvitka_adr, bsend:=((fb_su3_pidsvitka_send.bData XOR fb_su3_pidsvitka_read.bData XOR su3_pidsvitka)OR fb_heartbeat_timer.q));
IF NOT fb_su3_pidsvitka_read.bDataReceive OR  fb_heartbeat_timer.q THEN fb_su3_pidsvitka_send.bSend:=FALSE; fb_su3_pidsvitka_send(str_Rec:=fb_KL6301_0.str_Data_Rec, bData:=su3_pidsvitka,  Group_Address:=su3_pidsvitka_adr);END_IF
fb_su3_bra_send(str_Rec:=fb_KL6301_0.str_Data_Rec, bData:=su3_bra,  Group_Address:=su3_bra_adr, bsend:=((fb_su3_bra_send.bData XOR fb_su3_bra_read.bData XOR su3_bra)OR fb_heartbeat_timer.q));
IF NOT fb_su3_bra_read.bDataReceive OR  fb_heartbeat_timer.q THEN fb_su3_bra_send.bSend:=FALSE; fb_su3_bra_send(str_Rec:=fb_KL6301_0.str_Data_Rec, bData:=su3_bra,  Group_Address:=su3_bra_adr);END_IF
fb_su3_kontrazhur_send(str_Rec:=fb_KL6301_0.str_Data_Rec, bData:=su3_kontrazhur,  Group_Address:=su3_kontrazhur_adr, bsend:=((fb_su3_kontrazhur_send.bData XOR fb_su3_kontrazhur_read.bData XOR su3_kontrazhur)OR fb_heartbeat_timer.q));
IF NOT fb_su3_kontrazhur_read.bDataReceive OR  fb_heartbeat_timer.q THEN fb_su3_kontrazhur_send.bSend:=FALSE; fb_su3_kontrazhur_send(str_Rec:=fb_KL6301_0.str_Data_Rec, bData:=su3_kontrazhur,  Group_Address:=su3_kontrazhur_adr);END_IF
fb_su3_kontrazhur_k_send(str_Rec:=fb_KL6301_0.str_Data_Rec, bData:=su3_kontrazhur_k,  Group_Address:=su3_kontrazhur_k_adr, bsend:=((fb_su3_kontrazhur_k_send.bData XOR fb_su3_kontrazhur_k_read.bData XOR su3_kontrazhur_k)OR fb_heartbeat_timer.q));
IF NOT fb_su3_kontrazhur_k_read.bDataReceive OR  fb_heartbeat_timer.q THEN fb_su3_kontrazhur_k_send.bSend:=FALSE; fb_su3_kontrazhur_k_send(str_Rec:=fb_KL6301_0.str_Data_Rec, bData:=su3_kontrazhur_k,  Group_Address:=su3_kontrazhur_k_adr);END_IF
fb_su3_lampa_send(str_Rec:=fb_KL6301_0.str_Data_Rec, bData:=su3_lampa,  Group_Address:=su3_lampa_adr, bsend:=((fb_su3_lampa_send.bData XOR fb_su3_lampa_read.bData XOR su3_lampa)OR fb_heartbeat_timer.q));
IF NOT fb_su3_lampa_read.bDataReceive OR  fb_heartbeat_timer.q THEN fb_su3_lampa_send.bSend:=FALSE; fb_su3_lampa_send(str_Rec:=fb_KL6301_0.str_Data_Rec, bData:=su3_lampa,  Group_Address:=su3_lampa_adr);END_IF
fb_dytjacha_send(str_Rec:=fb_KL6301_0.str_Data_Rec, bData:=dytjacha,  Group_Address:=dytjacha_adr, bsend:=((fb_dytjacha_send.bData XOR fb_dytjacha_read.bData XOR dytjacha)OR fb_heartbeat_timer.q));
IF NOT fb_dytjacha_read.bDataReceive OR  fb_heartbeat_timer.q THEN fb_dytjacha_send.bSend:=FALSE; fb_dytjacha_send(str_Rec:=fb_KL6301_0.str_Data_Rec, bData:=dytjacha,  Group_Address:=dytjacha_adr);END_IF
fb_dytjacha_bra_send(str_Rec:=fb_KL6301_0.str_Data_Rec, bData:=dytjacha_bra,  Group_Address:=dytjacha_bra_adr, bsend:=((fb_dytjacha_bra_send.bData XOR fb_dytjacha_bra_read.bData XOR dytjacha_bra)OR fb_heartbeat_timer.q));
IF NOT fb_dytjacha_bra_read.bDataReceive OR  fb_heartbeat_timer.q THEN fb_dytjacha_bra_send.bSend:=FALSE; fb_dytjacha_bra_send(str_Rec:=fb_KL6301_0.str_Data_Rec, bData:=dytjacha_bra,  Group_Address:=dytjacha_bra_adr);END_IF
fb_garderob_send(str_Rec:=fb_KL6301_0.str_Data_Rec, bData:=garderob,  Group_Address:=garderob_adr, bsend:=((fb_garderob_read.bData XOR garderob XOR fb_garderob_send.bData )OR fb_heartbeat_timer.q));
IF NOT fb_garderob_read.bDataReceive OR  fb_heartbeat_timer.q THEN fb_garderob_send.bSend:=FALSE; fb_garderob_send(str_Rec:=fb_KL6301_0.str_Data_Rec, bData:=garderob,  Group_Address:=garderob_adr);END_IF
fb_bar_send(str_Rec:=fb_KL6301_0.str_Data_Rec, bData:=bar,  Group_Address:=bar_adr, bsend:=((fb_bar_send.bData XOR fb_bar_read.bData XOR bar)OR fb_heartbeat_timer.q));
IF NOT fb_bar_read.bDataReceive OR  fb_heartbeat_timer.q THEN fb_bar_send.bSend:=FALSE; fb_bar_send(str_Rec:=fb_KL6301_0.str_Data_Rec, bData:=bar,  Group_Address:=bar_adr);END_IF
fb_korydor_skeli_send(str_Rec:=fb_KL6301_0.str_Data_Rec, bData:=korydor_skeli,  Group_Address:=korydor_skeli_adr, bsend:=((fb_korydor_skeli_read.bData XOR korydor_skeli XOR fb_korydor_skeli_send.bData )OR fb_heartbeat_timer.q));
IF  NOT fb_korydor_skeli_read.bDataReceive OR  fb_heartbeat_timer.q THEN  fb_korydor_skeli_send.bSend:=FALSE; fb_korydor_skeli_send(str_Rec:=fb_KL6301_0.str_Data_Rec, bData:=korydor_skeli,  Group_Address:=korydor_skeli_adr);END_IF
fb_choven_send(str_Rec:=fb_KL6301_0.str_Data_Rec, bData:=choven,  Group_Address:=choven_adr, bsend:=((fb_choven_read.bData XOR choven XOR fb_choven_send.bData )OR fb_heartbeat_timer.q));
IF NOT fb_choven_read.bDataReceive OR  fb_heartbeat_timer.q THEN fb_choven_send.bSend:=FALSE; fb_choven_send(str_Rec:=fb_KL6301_0.str_Data_Rec, bData:=choven,  Group_Address:=choven_adr);END_IF
fb_korydor_svitlo_send(str_Rec:=fb_KL6301_0.str_Data_Rec, bData:=korydor_svitlo,  Group_Address:=korydor_svitlo_adr, bsend:=((fb_korydor_svitlo_send.bData XOR fb_korydor_svitlo_read.bData XOR korydor_svitlo)OR fb_heartbeat_timer.q));
IF NOT fb_korydor_svitlo_read.bDataReceive OR  fb_heartbeat_timer.q THEN fb_korydor_svitlo_send.bSend:=FALSE; fb_korydor_svitlo_send(str_Rec:=fb_KL6301_0.str_Data_Rec, bData:=korydor_svitlo,  Group_Address:=korydor_svitlo_adr);END_IF
fb_korydor_lampa_send(str_Rec:=fb_KL6301_0.str_Data_Rec, bData:=korydor_lampa,  Group_Address:=korydor_lampa_adr, bsend:=((fb_korydor_lampa_read.bData XOR korydor_lampa XOR fb_korydor_lampa_send.bData )OR fb_heartbeat_timer.q));
IF NOT fb_korydor_lampa_read.bDataReceive OR  fb_heartbeat_timer.q THEN fb_korydor_lampa_send.bSend:=FALSE; fb_korydor_lampa_send(str_Rec:=fb_KL6301_0.str_Data_Rec, bData:=korydor_lampa,  Group_Address:=korydor_lampa_adr);END_IF
fb_serverna_send(str_Rec:=fb_KL6301_0.str_Data_Rec, bData:=serverna,  Group_Address:=serverna_adr, bsend:=((fb_serverna_send.bData XOR fb_serverna_read.bData XOR serverna)OR fb_heartbeat_timer.q));
IF NOT fb_serverna_read.bDataReceive OR  fb_heartbeat_timer.q THEN fb_serverna_send.bSend:=FALSE; fb_serverna_send(str_Rec:=fb_KL6301_0.str_Data_Rec, bData:=serverna,  Group_Address:=serverna_adr);END_IF
END_ACTION
ACTION PanelBus:
CASE fb_kl6301_0.GroupReceive.SUB_MAIN OF
	1:(*vitalnya*)
	IF fb_kl6301_0.GroupReceive.number <10 AND fb_kl6301_0.GroupReceive.number <>0 THEN vitalnya_hvac.heat_mode:=fb_kl6301_0.GroupReceive.number;END_IF
		CASE fb_kl6301_0.GroupReceive.number OF
			0:		fb_temp_read(Group_Address:=vitalnya_T_EIB_addr, strData_Rec:=fb_KL6301_0.str_Data_Rec, rData=>Vitalnya_HVAC.cur_t); (*temperature*)
			1:		fb_setpoint_read(Group_address:=vitalnya_cooling_EIB_addr, strData_Rec:=fb_KL6301_0.str_Data_Rec, byData=>setpoint_vitalnya_dpt4 ); (*cooling*)
					CASE REAL_TO_INT(setpoint_vitalnya_dpt4*100/255.0) OF
						0..30:		vitalnya_hvac.heat_speed:=1;
									vitalnya_hvac.t_ust_cool:= REAL_TO_INT(setpoint_vitalnya_dpt4*100/255.0); (*low speed*)
						31..59:		vitalnya_hvac.heat_speed:=2;
									vitalnya_hvac.t_ust_cool:= REAL_TO_INT(setpoint_vitalnya_dpt4*100/255.0-30); (*med speed*)
						60..100:	vitalnya_hvac.heat_speed:=3;
									vitalnya_hvac.t_ust_cool:= REAL_TO_INT(setpoint_vitalnya_dpt4*100/255.0-60); (*high speed*)
					END_CASE
					vitalnya_hvac.cur_t_ust:=vitalnya_hvac.t_ust_cool;
					(*
					надсилання в мережу прийнятого значення завдання
					fb_actual_setpoint_send(group_address:=vitalnya_actual_setpoint_addr, str_Rec:=fb_kl6301_0.str_Data_Rec, rData:=vitalnya_hvac.cur_t_ust);
					*)
			2:		fb_setpoint_read(Group_address:=vitalnya_heating_EIB_addr, strData_Rec:=fb_KL6301_0.str_Data_Rec, byData=>setpoint_vitalnya_dpt4 );  (*heating*)
					CASE REAL_TO_INT(setpoint_vitalnya_dpt4*100/255.0) OF
						0..30:		vitalnya_hvac.heat_speed:=1;
									vitalnya_hvac.t_ust_heat:= REAL_TO_INT(setpoint_vitalnya_dpt4*100/255.0); (*low speed*)
						31..59:		vitalnya_hvac.heat_speed:=2;
									vitalnya_hvac.t_ust_heat:= REAL_TO_INT(setpoint_vitalnya_dpt4*100/255.0-30); (*med speed*)
						60..100:	vitalnya_hvac.heat_speed:=3;
									vitalnya_hvac.t_ust_heat:= REAL_TO_INT(setpoint_vitalnya_dpt4*100/255.0-60); (*high speed*)
					END_CASE
					vitalnya_hvac.cur_t_ust:=vitalnya_hvac.t_ust_heat;
					(*
					fb_actual_setpoint_send(group_address:=vitalnya_actual_setpoint_addr, str_Rec:=fb_kl6301_0.str_Data_Rec, rData:=vitalnya_hvac.cur_t_ust);
					*)
			3:		fb_setpoint_read(Group_address:=vitalnya_fan_EIB_addr, strData_Rec:=fb_KL6301_0.str_Data_Rec, byData=>fanspeed_dpt4);
					VITALNYA_HVAC.heat_speed:=REAL_TO_USINT(fanspeed_dpt4*100/255.0);
			4:		VITALNYA_HVAC.heat_mode:=0;
			5:		fb_actual_setpoint_read(Group_Address:=vitalnya_actual_setpoint_addr, strData_Rec:=fb_KL6301_0.str_Data_Rec );
					vitalnya_hvac.cur_t_ust:=fb_actual_setpoint_read.rData;
		END_CASE;
	2: ;(*kino*)
	IF fb_kl6301_0.GroupReceive.number <10 AND fb_kl6301_0.GroupReceive.number <>0 THEN kino_hvac.heat_mode:=fb_kl6301_0.GroupReceive.number;END_IF
		CASE fb_kl6301_0.GroupReceive.number OF
			0:		fb_temp_read(Group_Address:=kino_T_EIB_addr, strData_Rec:=fb_KL6301_0.str_Data_Rec, rData=>kino_HVAC.cur_t); (*temperature*)
			1:		fb_setpoint_read(Group_address:=kino_cooling_EIB_addr, strData_Rec:=fb_KL6301_0.str_Data_Rec, byData=>setpoint_kino_dpt4 ); (*cooling*)
					CASE REAL_TO_INT(setpoint_kino_dpt4*100/255.0) OF
						0..30:		kino_hvac.heat_speed:=1;
									kino_hvac.t_ust_cool:= REAL_TO_INT(setpoint_kino_dpt4*100/255.0); (*low speed*)
						31..59:		kino_hvac.heat_speed:=2;
									kino_hvac.t_ust_cool:= REAL_TO_INT(setpoint_kino_dpt4*100/255.0-30); (*med speed*)
						60..100:	kino_hvac.heat_speed:=3;
									kino_hvac.t_ust_cool:= REAL_TO_INT(setpoint_kino_dpt4*100/255.0-60); (*high speed*)
					END_CASE
					kino_hvac.cur_t_ust:=kino_hvac.t_ust_cool;
					(*fb_actual_setpoint_send(group_address:=kino_actual_setpoint_addr, str_Rec:=fb_kl6301_0.str_Data_Rec, rData:=kino_hvac.cur_t_ust);*)
					kino_HVAc.manual_mode:=0;

			2:		fb_setpoint_read(Group_address:=kino_heating_EIB_addr, strData_Rec:=fb_KL6301_0.str_Data_Rec, byData=>setpoint_kino_dpt4 );  (*heating*)
					CASE REAL_TO_INT(setpoint_kino_dpt4*100/255.0) OF
						0..30:		kino_hvac.heat_speed:=1;
									kino_hvac.t_ust_heat:= REAL_TO_INT(setpoint_kino_dpt4*100/255.0); (*low speed*)
						31..59:		kino_hvac.heat_speed:=2;
									kino_hvac.t_ust_heat:= REAL_TO_INT(setpoint_kino_dpt4*100/255.0-30); (*med speed*)
						60..100:	kino_hvac.heat_speed:=3;
									kino_hvac.t_ust_heat:= REAL_TO_INT(setpoint_kino_dpt4*100/255.0-60); (*high speed*)
					END_CASE
					kino_hvac.cur_t_ust:=kino_hvac.t_ust_heat;
					(*fb_actual_setpoint_send(group_address:=kino_actual_setpoint_addr, str_Rec:=fb_kl6301_0.str_Data_Rec, rData:=kino_hvac.cur_t_ust);*)
					kino_HVAc.manual_mode:=0;
			3:		fb_setpoint_read(Group_address:=kino_fan_EIB_addr, strData_Rec:=fb_KL6301_0.str_Data_Rec, byData=>fanspeed_dpt4);
					kino_HVAC.heat_speed:=REAL_TO_USINT(fanspeed_dpt4*100/255.0);
					kino_HVAc.manual_mode:=0;
			4:		KINO_HVAC .heat_mode:=0; kino_HVAc.manual_mode:=1;
			5:		fb_actual_setpoint_read(Group_Address:=kino_actual_setpoint_addr, strData_Rec:=fb_KL6301_0.str_Data_Rec );
					kino_hvac.cur_t_ust:=fb_actual_setpoint_read.rData;
					kino_HVAc.manual_mode:=0;

		END_CASE;

	3: ;(*studio*)
	IF fb_kl6301_0.GroupReceive.number <10 AND fb_kl6301_0.GroupReceive.number <>0 THEN studio_hvac.heat_mode:=fb_kl6301_0.GroupReceive.number;END_IF
		CASE fb_kl6301_0.GroupReceive.number OF
			0:		fb_temp_read(Group_Address:=studio_T_EIB_addr, strData_Rec:=fb_KL6301_0.str_Data_Rec, rData=>studio_HVAC.cur_t); (*temperature*)
			1:		fb_setpoint_read(Group_address:=studio_cooling_EIB_addr, strData_Rec:=fb_KL6301_0.str_Data_Rec, byData=>setpoint_studio_dpt4 ); (*cooling*)
					CASE REAL_TO_INT(setpoint_studio_dpt4*100/255.0) OF
						0..30:		studio_hvac.heat_speed:=1;
									studio_hvac.t_ust_cool:= REAL_TO_INT(setpoint_studio_dpt4*100/255.0); (*low speed*)
						31..59:		studio_hvac.heat_speed:=2;
									studio_hvac.t_ust_cool:= REAL_TO_INT(setpoint_studio_dpt4*100/255.0-30); (*med speed*)
						60..100:	studio_hvac.heat_speed:=3;
									studio_hvac.t_ust_cool:= REAL_TO_INT(setpoint_studio_dpt4*100/255.0-60); (*high speed*)
					END_CASE
					studio_hvac.cur_t_ust:=studio_hvac.t_ust_cool;
					(*fb_actual_setpoint_send(group_address:=studio_actual_setpoint_addr, str_Rec:=fb_kl6301_0.str_Data_Rec, rData:=studio_hvac.cur_t_ust);*)

			2:		fb_setpoint_read(Group_address:=studio_heating_EIB_addr, strData_Rec:=fb_KL6301_0.str_Data_Rec, byData=>setpoint_studio_dpt4 );  (*heating*)
					CASE REAL_TO_INT(setpoint_studio_dpt4*100/255.0) OF
						0..30:		studio_hvac.heat_speed:=1;
									studio_hvac.t_ust_heat:= REAL_TO_INT(setpoint_studio_dpt4*100/255.0); (*low speed*)
						31..59:		studio_hvac.heat_speed:=2;
									studio_hvac.t_ust_heat:= REAL_TO_INT(setpoint_studio_dpt4*100/255.0-30); (*med speed*)
						60..100:	studio_hvac.heat_speed:=3;
									studio_hvac.t_ust_heat:= REAL_TO_INT(setpoint_studio_dpt4*100/255.0-60); (*high speed*)
					END_CASE
					studio_hvac.cur_t_ust:=studio_hvac.t_ust_heat;
					(*fb_actual_setpoint_send(group_address:=studio_actual_setpoint_addr, str_Rec:=fb_kl6301_0.str_Data_Rec, rData:=studio_hvac.cur_t_ust);*)

			3:		fb_setpoint_read(Group_address:=studio_fan_EIB_addr, strData_Rec:=fb_KL6301_0.str_Data_Rec, byData=>fanspeed_dpt4);
					studio_HVAC.heat_speed:=REAL_TO_USINT(fanspeed_dpt4*100/255.0);
			4:		STUDIO_HVAC.heat_mode:=0;
			5:		fb_actual_setpoint_read(Group_Address:=studio_actual_setpoint_addr, strData_Rec:=fb_KL6301_0.str_Data_Rec );
					studio_hvac.cur_t_ust:=fb_actual_setpoint_read.rData;

		END_CASE;

	4: ;(*kabinet*)
		IF fb_kl6301_0.GroupReceive.number <10 AND fb_kl6301_0.GroupReceive.number <>0 THEN kabinet_hvac.heat_mode:=fb_kl6301_0.GroupReceive.number;END_IF
		CASE fb_kl6301_0.GroupReceive.number OF
			0:		fb_temp_read(Group_Address:=kabinet_T_EIB_addr, strData_Rec:=fb_KL6301_0.str_Data_Rec, rData=>kabinet_HVAC.cur_t); (*temperature*)
			1:		fb_setpoint_read(Group_address:=kabinet_cooling_EIB_addr, strData_Rec:=fb_KL6301_0.str_Data_Rec, byData=>setpoint_kabinet_dpt4 ); (*cooling*)
					CASE REAL_TO_INT(setpoint_kabinet_dpt4*100/255.0) OF
						0..30:		kabinet_hvac.heat_speed:=1;
									kabinet_hvac.t_ust_cool:= REAL_TO_INT(setpoint_kabinet_dpt4*100/255.0); (*low speed*)
						31..59:		kabinet_hvac.heat_speed:=2;
									kabinet_hvac.t_ust_cool:= REAL_TO_INT(setpoint_kabinet_dpt4*100/255.0-30); (*med speed*)
						60..100:	kabinet_hvac.heat_speed:=3;
									kabinet_hvac.t_ust_cool:= REAL_TO_INT(setpoint_kabinet_dpt4*100/255.0-60); (*high speed*)
					END_CASE
					kabinet_hvac.cur_t_ust:=kabinet_hvac.t_ust_cool;
					(*fb_actual_setpoint_send(group_address:=kabinet_actual_setpoint_addr, str_Rec:=fb_kl6301_0.str_Data_Rec, rData:=kabinet_hvac.cur_t_ust);*)

			2:		fb_setpoint_read(Group_address:=kabinet_heating_EIB_addr, strData_Rec:=fb_KL6301_0.str_Data_Rec, byData=>setpoint_kabinet_dpt4 );  (*heating*)
					CASE REAL_TO_INT(setpoint_kabinet_dpt4*100/255.0) OF
						0..30:		kabinet_hvac.heat_speed:=1;
									kabinet_hvac.t_ust_heat:= REAL_TO_INT(setpoint_kabinet_dpt4*100/255.0); (*low speed*)
						31..59:		kabinet_hvac.heat_speed:=2;
									kabinet_hvac.t_ust_heat:= REAL_TO_INT(setpoint_kabinet_dpt4*100/255.0-30); (*med speed*)
						60..100:	kabinet_hvac.heat_speed:=3;
									kabinet_hvac.t_ust_heat:= REAL_TO_INT(setpoint_kabinet_dpt4*100/255.0-60); (*high speed*)
					END_CASE
					kabinet_hvac.cur_t_ust:=kabinet_hvac.t_ust_heat;
					(*fb_actual_setpoint_send(group_address:=kabinet_actual_setpoint_addr, str_Rec:=fb_kl6301_0.str_Data_Rec, rData:=kabinet_hvac.cur_t_ust);*)


			3:		fb_setpoint_read(Group_address:=kabinet_fan_EIB_addr, strData_Rec:=fb_KL6301_0.str_Data_Rec, byData=>fanspeed_dpt4);
					kabinet_HVAC.heat_speed:=REAL_TO_USINT(fanspeed_dpt4*100/255.0);
			4:		KABINET_HVAC.heat_mode:=0;
			5:		fb_actual_setpoint_read(Group_Address:=kabinet_actual_setpoint_addr, strData_Rec:=fb_KL6301_0.str_Data_Rec );
					kabinet_hvac.cur_t_ust:=fb_actual_setpoint_read.rData;

		END_CASE;

	5: ;(*dytjacha*)
		IF fb_kl6301_0.GroupReceive.number <10 AND fb_kl6301_0.GroupReceive.number <>0 THEN dytjacha_hvac.heat_mode:=fb_kl6301_0.GroupReceive.number;END_IF
		CASE fb_kl6301_0.GroupReceive.number OF
			0:		fb_temp_read(Group_Address:=dytjacha_T_EIB_addr, strData_Rec:=fb_KL6301_0.str_Data_Rec, rData=>dytjacha_HVAC.cur_t); (*temperature*)
			1:		fb_setpoint_read(Group_address:=dytjacha_cooling_EIB_addr, strData_Rec:=fb_KL6301_0.str_Data_Rec, byData=>setpoint_dytjacha_dpt4 ); (*cooling*)
					CASE REAL_TO_INT(setpoint_dytjacha_dpt4*100/255.0) OF
						0..30:		dytjacha_hvac.heat_speed:=1;
									dytjacha_hvac.t_ust_cool:= REAL_TO_INT(setpoint_dytjacha_dpt4*100/255.0); (*low speed*)
						31..59:		dytjacha_hvac.heat_speed:=2;
									dytjacha_hvac.t_ust_cool:= REAL_TO_INT(setpoint_dytjacha_dpt4*100/255.0-30); (*med speed*)
						60..100:	dytjacha_hvac.heat_speed:=3;
									dytjacha_hvac.t_ust_cool:= REAL_TO_INT(setpoint_dytjacha_dpt4*100/255.0-60); (*high speed*)
					END_CASE
					dytjacha_hvac.cur_t_ust:=dytjacha_hvac.t_ust_cool;
					(*fb_actual_setpoint_send(group_address:=dytjacha_actual_setpoint_addr, str_Rec:=fb_kl6301_0.str_Data_Rec, rData:=dytjacha_hvac.cur_t_ust);*)

			2:		fb_setpoint_read(Group_address:=dytjacha_heating_EIB_addr, strData_Rec:=fb_KL6301_0.str_Data_Rec, byData=>setpoint_dytjacha_dpt4 );  (*heating*)
					CASE REAL_TO_INT(setpoint_dytjacha_dpt4*100/255.0) OF
						0..30:		dytjacha_hvac.heat_speed:=1;
									dytjacha_hvac.t_ust_heat:= REAL_TO_INT(setpoint_dytjacha_dpt4*100/255.0); (*low speed*)
						31..59:		dytjacha_hvac.heat_speed:=2;
									dytjacha_hvac.t_ust_heat:= REAL_TO_INT(setpoint_dytjacha_dpt4*100/255.0-30); (*med speed*)
						60..100:	dytjacha_hvac.heat_speed:=3;
									dytjacha_hvac.t_ust_heat:= REAL_TO_INT(setpoint_dytjacha_dpt4*100/255.0-60); (*high speed*)
					END_CASE
					dytjacha_hvac.cur_t_ust:=dytjacha_hvac.t_ust_heat;
					(*fb_actual_setpoint_send(group_address:=dytjacha_actual_setpoint_addr, str_Rec:=fb_kl6301_0.str_Data_Rec, rData:=dytjacha_hvac.cur_t_ust);*)


			3:		fb_setpoint_read(Group_address:=dytjacha_fan_EIB_addr, strData_Rec:=fb_KL6301_0.str_Data_Rec, byData=>fanspeed_dpt4);
					dytjacha_HVAC.heat_speed:=REAL_TO_USINT(fanspeed_dpt4*100/255.0);
			4:		DYTJACHA_HVAC.heat_mode:=0;
			5:		fb_actual_setpoint_read(Group_Address:=dytjacha_actual_setpoint_addr, strData_Rec:=fb_KL6301_0.str_Data_Rec );
					dytjacha_hvac.cur_t_ust:=fb_actual_setpoint_read.rData;

		END_CASE;

	6: ;(*spalnya*)
		IF fb_kl6301_0.GroupReceive.number <10 AND fb_kl6301_0.GroupReceive.number <>0 THEN spalnya_hvac.heat_mode:=fb_kl6301_0.GroupReceive.number;END_IF
		CASE fb_kl6301_0.GroupReceive.number OF
			0:		fb_temp_read(Group_Address:=spalnya_T_EIB_addr, strData_Rec:=fb_KL6301_0.str_Data_Rec, rData=>spalnya_HVAC.cur_t); (*temperature*)
			1:		fb_setpoint_read(Group_address:=spalnya_cooling_EIB_addr, strData_Rec:=fb_KL6301_0.str_Data_Rec, byData=>setpoint_spalnya_dpt4 ); (*cooling*)
					CASE REAL_TO_INT(setpoint_spalnya_dpt4*100/255.0) OF
						0..30:		spalnya_hvac.heat_speed:=1;
									spalnya_hvac.t_ust_cool:= REAL_TO_INT(setpoint_spalnya_dpt4*100/255.0); (*low speed*)
						31..59:		spalnya_hvac.heat_speed:=2;
									spalnya_hvac.t_ust_cool:= REAL_TO_INT(setpoint_spalnya_dpt4*100/255.0-30); (*med speed*)
						60..100:	spalnya_hvac.heat_speed:=3;
									spalnya_hvac.t_ust_cool:= REAL_TO_INT(setpoint_spalnya_dpt4*100/255.0-60); (*high speed*)
					END_CASE
					spalnya_hvac.cur_t_ust:=spalnya_hvac.t_ust_cool;
					(*fb_actual_setpoint_send(group_address:=spalnya_actual_setpoint_addr, str_Rec:=fb_kl6301_0.str_Data_Rec, rData:=spalnya_hvac.cur_t_ust);*)

			2:		fb_setpoint_read(Group_address:=spalnya_heating_EIB_addr, strData_Rec:=fb_KL6301_0.str_Data_Rec, byData=>setpoint_spalnya_dpt4 );  (*heating*)
					CASE REAL_TO_INT(setpoint_spalnya_dpt4*100/255.0) OF
						0..30:		spalnya_hvac.heat_speed:=1;
									spalnya_hvac.t_ust_heat:= REAL_TO_INT(setpoint_spalnya_dpt4*100/255.0); (*low speed*)
						31..59:		spalnya_hvac.heat_speed:=2;
									spalnya_hvac.t_ust_heat:= REAL_TO_INT(setpoint_spalnya_dpt4*100/255.0-30); (*med speed*)
						60..100:	spalnya_hvac.heat_speed:=3;
									spalnya_hvac.t_ust_heat:= REAL_TO_INT(setpoint_spalnya_dpt4*100/255.0-60); (*high speed*)
					END_CASE
					spalnya_hvac.cur_t_ust:=spalnya_hvac.t_ust_heat;
					(*fb_actual_setpoint_send(group_address:=spalnya_actual_setpoint_addr, str_Rec:=fb_kl6301_0.str_Data_Rec, rData:=spalnya_hvac.cur_t_ust);*)


			3:		fb_setpoint_read(Group_address:=spalnya_fan_EIB_addr, strData_Rec:=fb_KL6301_0.str_Data_Rec, byData=>fanspeed_dpt4);
					spalnya_HVAC.heat_speed:=REAL_TO_USINT(fanspeed_dpt4*100/255.0);
			4:		SPALNYA_HVAC.heat_mode:=0;
			5:		fb_actual_setpoint_read(Group_Address:=spalnya_actual_setpoint_addr, strData_Rec:=fb_KL6301_0.str_Data_Rec );
					spalnya_hvac.cur_t_ust:=fb_actual_setpoint_read.rData;

		END_CASE;
END_CASE



(*hdl gate can transmit 2byte values, but they can not be assigned to DLP panel AC unit setpoint value directly,
so for every setpoint value in range [20,30] a 1 bit eib telegram with corresponding  adress +100 ( [120,130] ) should be generated and transmitted to HDL logic module and then
logic module assigns it to apropriate value DLP panel AC unit. 
amen*)
fb_setpoint_switch_send.iMode:=2;
fb_setpoint_switch_send.bStart:=TRUE;
IF vitalnya_hvac.cur_t_ust_prev <> vitalnya_hvac.cur_t_ust THEN
	fb_setpoint_switch_send.Group_Address.NUMBER:=REAL_TO_BYTE(vitalnya_hvac.cur_t_ust)+100;
	fb_setpoint_switch_send.Group_Address.MAIN:=1;
	fb_setpoint_switch_send.Group_Address.SUB_MAIN:=1;
	fb_setpoint_switch_send(str_Rec:=fb_KL6301_0.str_Data_Rec, bData:=FALSE);
	fb_setpoint_switch_send(str_Rec:=fb_KL6301_0.str_Data_Rec, bData:=TRUE);
END_IF
IF kino_hvac.cur_t_ust_prev <> kino_hvac.cur_t_ust THEN
	fb_setpoint_switch_send.Group_Address.NUMBER:=REAL_TO_BYTE(kino_hvac.cur_t_ust)+100;
	fb_setpoint_switch_send.Group_Address.MAIN:=1;
	fb_setpoint_switch_send.Group_Address.SUB_MAIN:=2;
	fb_setpoint_switch_send(str_Rec:=fb_KL6301_0.str_Data_Rec, bData:=1);
	fb_setpoint_switch_send(str_Rec:=fb_KL6301_0.str_Data_Rec, bData:=0);
END_IF
IF studio_hvac.cur_t_ust_prev <> studio_hvac.cur_t_ust THEN
	fb_setpoint_switch_send.Group_Address.NUMBER:=REAL_TO_BYTE(studio_hvac.cur_t_ust)+100;
	fb_setpoint_switch_send.Group_Address.MAIN:=1;
	fb_setpoint_switch_send.Group_Address.SUB_MAIN:=3;
	fb_setpoint_switch_send(str_Rec:=fb_KL6301_0.str_Data_Rec, bData:=1);
	fb_setpoint_switch_send(str_Rec:=fb_KL6301_0.str_Data_Rec, bData:=0);
END_IF
IF kabinet_hvac.cur_t_ust_prev <> kabinet_hvac.cur_t_ust THEN
	fb_setpoint_switch_send.Group_Address.NUMBER:=REAL_TO_BYTE(kabinet_hvac.cur_t_ust)+100;
	fb_setpoint_switch_send.Group_Address.MAIN:=1;
	fb_setpoint_switch_send.Group_Address.SUB_MAIN:=4;
	fb_setpoint_switch_send(str_Rec:=fb_KL6301_0.str_Data_Rec, bData:=1);
	fb_setpoint_switch_send(str_Rec:=fb_KL6301_0.str_Data_Rec, bData:=0);
END_IF
IF dytjacha_hvac.cur_t_ust_prev <> dytjacha_hvac.cur_t_ust THEN
	fb_setpoint_switch_send.Group_Address.NUMBER:=REAL_TO_BYTE(dytjacha_hvac.cur_t_ust)+100;
	fb_setpoint_switch_send.Group_Address.MAIN:=1;
	fb_setpoint_switch_send.Group_Address.SUB_MAIN:=5;
	fb_setpoint_switch_send(str_Rec:=fb_KL6301_0.str_Data_Rec, bData:=1);
	fb_setpoint_switch_send(str_Rec:=fb_KL6301_0.str_Data_Rec, bData:=0);
END_IF
IF spalnya_hvac.cur_t_ust_prev <> spalnya_hvac.cur_t_ust THEN
	fb_setpoint_switch_send.Group_Address.NUMBER:=REAL_TO_BYTE(spalnya_hvac.cur_t_ust)+100;
	fb_setpoint_switch_send.Group_Address.MAIN:=1;
	fb_setpoint_switch_send.Group_Address.SUB_MAIN:=6;
	fb_setpoint_switch_send(str_Rec:=fb_KL6301_0.str_Data_Rec, bData:=1);
	fb_setpoint_switch_send(str_Rec:=fb_KL6301_0.str_Data_Rec, bData:=0);
END_IF
END_ACTION
ACTION timers:
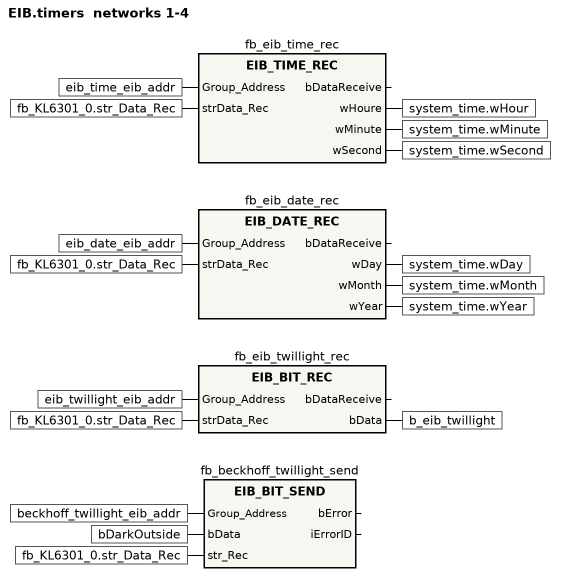
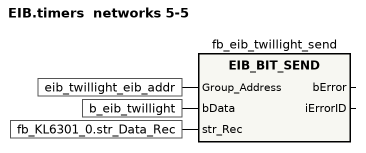
_FBD_ (* Function Block Diagram *)
NETWORK 1
	fb_eib_time_rec:EIB_TIME_REC(Group_Address: eib_time_eib_addr, strData_Rec: fb_KL6301_0.str_Data_Rec, wHoure => system_time.wHour, wMinute => system_time.wMinute, wSecond => system_time.wSecond)
NETWORK 2
	fb_eib_date_rec:EIB_DATE_REC(Group_Address: eib_date_eib_addr, strData_Rec: fb_KL6301_0.str_Data_Rec, wDay => system_time.wDay, wMonth => system_time.wMonth, wYear => system_time.wYear)
NETWORK 3
	fb_eib_twillight_rec:EIB_BIT_REC(Group_Address: eib_twillight_eib_addr, strData_Rec: fb_KL6301_0.str_Data_Rec, bData => b_eib_twillight)
NETWORK 4
	fb_beckhoff_twillight_send:EIB_BIT_SEND(Group_Address: beckhoff_twillight_eib_addr, bData: bDarkOutside, str_Rec: fb_KL6301_0.str_Data_Rec)
NETWORK 5
	fb_eib_twillight_send:EIB_BIT_SEND(Group_Address: eib_twillight_eib_addr, bData: b_eib_twillight, str_Rec: fb_KL6301_0.str_Data_Rec)
_END_FBD_
(* the same logic as Structured Text *)
(* Network 1 *)
fb_eib_time_rec(Group_Address := eib_time_eib_addr, strData_Rec := fb_KL6301_0.str_Data_Rec);
system_time.wHour := fb_eib_time_rec.wHoure;
system_time.wMinute := fb_eib_time_rec.wMinute;
system_time.wSecond := fb_eib_time_rec.wSecond;
(* Network 2 *)
fb_eib_date_rec(Group_Address := eib_date_eib_addr, strData_Rec := fb_KL6301_0.str_Data_Rec);
system_time.wDay := fb_eib_date_rec.wDay;
system_time.wMonth := fb_eib_date_rec.wMonth;
system_time.wYear := fb_eib_date_rec.wYear;
(* Network 3 *)
fb_eib_twillight_rec(Group_Address := eib_twillight_eib_addr, strData_Rec := fb_KL6301_0.str_Data_Rec);
b_eib_twillight := fb_eib_twillight_rec.bData;
(* Network 4 *)
fb_beckhoff_twillight_send(Group_Address := beckhoff_twillight_eib_addr, bData := bDarkOutside, str_Rec := fb_KL6301_0.str_Data_Rec);
(* Network 5 *)
fb_eib_twillight_send(Group_Address := eib_twillight_eib_addr, bData := b_eib_twillight, str_Rec := fb_KL6301_0.str_Data_Rec);
END_ACTION

(* POU RANGE_TO_RANGE, ST *)
FUNCTION RANGE_TO_RANGE : INT
VAR_INPUT
	by_input:BYTE;
	in_low_value: INT;
	in_high_value:INT;
	out_low_value: INT;
	out_high_value:INT;
END_VAR
VAR
	r_res: REAL;
	r_input: REAL;
END_VAR
r_input:=BYTE_TO_REAL(by_input);
IF out_high_value>out_low_value THEN
	r_res:=r_input/(in_high_value - in_low_value)*(out_high_value - out_low_value);
ELSE
	r_res:=out_low_value - (r_input / (in_high_value - in_low_value)*(out_low_value - out_high_value));
END_IF
RANGE_TO_RANGE:=REAL_TO_INT(r_res);
END_FUNCTION

(* POU GREATEST_OF, ST *)
FUNCTION GREATEST_OF : REAL
VAR_INPUT
	r_in1,r_in2:REAL;
END_VAR
VAR
END_VAR
IF r_in1>=r_in2 THEN
	GREATEST_OF:=r_in1;
ELSE
	GREATEST_OF:=r_in2;
END_IF
END_FUNCTION

(* POU ADS_write, ST *)
PROGRAM ADS_write
VAR
	write_timeout: TIME;
	b_write1, b_write2: BOOL;
	write_ads1, write_ads2, write_ads4: ADSWRITE;

	timer1, timer2:TP;
	errorcounter1, errorcounter2, pack_c:CTU ;
	test_word: WORD;
	i2,j2,i1,j1, i4,j4: INT;
	data_changed: BOOL;
	try_again2, try_again1, try_again4: BOOL;
	timer4: TP;
	b_write4: BOOL;
	errorcounter4: CTU;
END_VAR
write_timeout:=t#3s;

timer2(PT:=write_timeout*2);
timer2.IN:=FALSE;



FOR 2i:=0 TO (SIZEOF(data2floor))-1 DO
	IF data2floor[i2]<>data2floor_prev[i2]  OR try_again2 THEN
		b_write2:=TRUE;
		EXIT;
	ELSE
		b_write2:=FALSE;
	END_IF
END_FOR


FOR i1:=0 TO (SIZEOF(data1floor))-1 DO
	IF data1floor[i1]<>data1floor_prev[i1]  OR try_again1 THEN
		b_write1:=TRUE;
		EXIT;
	ELSE
		b_write1:=FALSE;
	END_IF
END_FOR


FOR i4:=0 TO (SIZEOF(data_derevo))-1 DO
	IF data_derevo[i4]<>data_derevo[i4]  OR try_again4 THEN
		b_write4:=TRUE;
		EXIT;
	ELSE
		b_write4:=FALSE;
	END_IF
END_FOR



(*
IF write_ads2.BUSY THEN b_write2:=FALSE; END_IF

	write_ads2(
		NETID:=ads_adr2,
		PORT:=800,
		IDXGRP:=16#4020,
		IDXOFFS:=300,
		WRITE:=b_write2,
		TMOUT:=write_timeout,
		LEN:=SIZEOF(data2floor),
		SRCADDR:=ADR(data2floor));
write_ads2.WRITE:=FALSE;

IF write_ads2.ERR AND NOT timer2.Q THEN
	timer2.IN:=TRUE;
	try_again2:=TRUE;
ELSE try_again2:=FALSE;
END_IF


(*1floor*)
FOR i1:=0 TO (SIZEOF(data1floor))-1 DO
	IF data1floor[i1]<>data1floor_prev[i1] AND NOT timer1.Q THEN
		b_write1:=TRUE;
		EXIT;
	ELSE
		b_write1:=FALSE;
	END_IF
END_FOR

IF try_again1 AND NOT timer1.Q THEN
	b_write1:=TRUE;
	try_again1:=FALSE;
END_IF

errorcounter1(cu:=write_ads1.ERR);

IF write_ads1.BUSY THEN b_write1:=FALSE; END_IF

	write_ads1(
		NETID:=ads_adr1,
		PORT:=800,
		IDXGRP:=16#4020,
		IDXOFFS:=300,
		WRITE:=b_write1,
		TMOUT:=write_timeout,
		LEN:=SIZEOF(data1floor),
		SRCADDR:=ADR(data1floor));

IF write_ads1.ERR AND NOT timer1.Q THEN
	timer1.IN:=TRUE;
	try_again1:=TRUE;
END_IF
timer1(PT:=write_timeout);
timer1.IN:=FALSE;



(*derevo*)
FOR i4:=0 TO (SIZEOF(data_derevo))-1 DO
	IF data_derevo[i4]<>data_derevo_prev[i4] AND NOT timer4.Q THEN
		b_write4:=TRUE;
		EXIT;
	ELSE
		b_write4:=FALSE;
	END_IF
END_FOR

IF try_again4 AND NOT timer4.Q THEN
	b_write4:=TRUE;
	try_again4:=FALSE;
END_IF

errorcounter4(cu:=write_ads4.ERR);


IF write_ads4.BUSY THEN b_write4:=FALSE; END_IF

	write_ads4(
		NETID:=ads_adr4,
		PORT:=800,
		IDXGRP:=16#4020,
		IDXOFFS:=400,
		WRITE:=b_write4,
		TMOUT:=write_timeout,
		LEN:=SIZEOF(data_derevo),
		SRCADDR:=ADR(data_derevo));

IF write_ads4.ERR AND NOT timer4.Q THEN
	timer4.IN:=TRUE;
	try_again4:=TRUE;
END_IF
timer4(PT:=write_timeout);
timer4.IN:=FALSE;
*)

FOR j1:=0 TO (SIZEOF(data1floor))-1 DO
	data1floor_prev[j1]:=data1floor[j1];
END_FOR

FOR j:=0 TO (SIZEOF(data2floor))-1 DO
	data2floor_prev[j]:=data2floor[j];
END_FOR

FOR j4:=0 TO (SIZEOF(data_derevo))-1 DO
	data_derevo_prev[j4]:=data_derevo[j4];
END_FOR
END_PROGRAM

(* POU ADS_Communication, CFC *)
PROGRAM ADS_Communication
VAR

	fb_floor1ADSwrite: ADSWRITE;
	fb_floor2ADSwrite: ADSWRITE;
	fb_floor4ADSwrite: ADSWRITE;


	counter_error,counter_busy: CTU;

	heartbeat:TP;
END_VAR
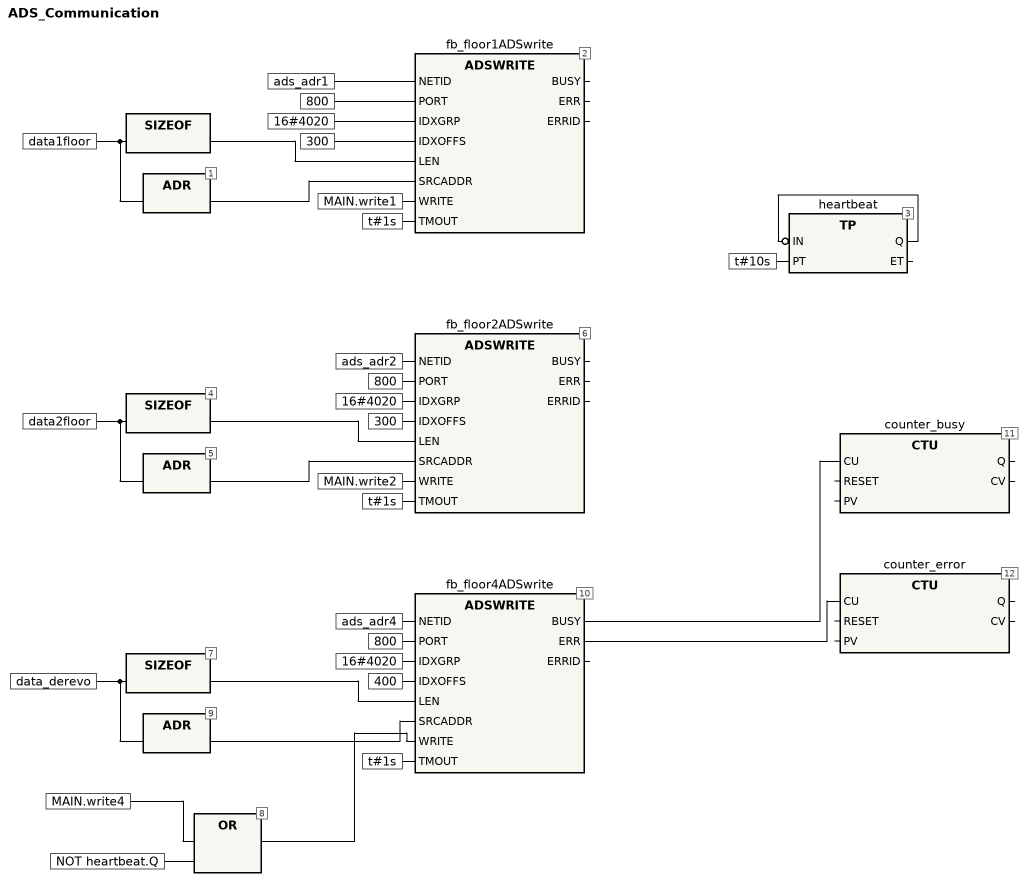
_CFC_ (* Continuous Function Chart, elements in execution order *)
#0 SIZEOF(data1floor)
#1 ADR(data1floor)
#2 fb_floor1ADSwrite:ADSWRITE(NETID: ads_adr1, PORT: 800, IDXGRP: 16#4020, IDXOFFS: 300, LEN: #0, SRCADDR: #1, WRITE: MAIN.write1, TMOUT: t#1s)
#3 heartbeat:TP(IN: NOT #3.Q, PT: t#10s)
#4 SIZEOF(data2floor)
#5 ADR(data2floor)
#6 fb_floor2ADSwrite:ADSWRITE(NETID: ads_adr2, PORT: 800, IDXGRP: 16#4020, IDXOFFS: 300, LEN: #4, SRCADDR: #5, WRITE: MAIN.write2, TMOUT: t#1s)
#7 SIZEOF(data_derevo)
#8 OR(MAIN.write4, NOT heartbeat.Q)
#9 ADR(data_derevo)
#10 fb_floor4ADSwrite:ADSWRITE(NETID: ads_adr4, PORT: 800, IDXGRP: 16#4020, IDXOFFS: 400, LEN: #7, SRCADDR: #9, WRITE: #8, TMOUT: t#1s)
#11 counter_busy:CTU(CU: #10.BUSY, RESET: -, PV: -)
#12 counter_error:CTU(CU: #10.ERR, RESET: -, PV: -)
_END_CFC_
(* the same logic as Structured Text *)
fb_floor1ADSwrite(NETID := ads_adr1, PORT := 800, IDXGRP := 16#4020, IDXOFFS := 300, LEN := SIZEOF(data1floor), SRCADDR := ADR(data1floor), WRITE := MAIN.write1, TMOUT := t#1s);
heartbeat(IN := NOT heartbeat.Q, PT := t#10s);
fb_floor2ADSwrite(NETID := ads_adr2, PORT := 800, IDXGRP := 16#4020, IDXOFFS := 300, LEN := SIZEOF(data2floor), SRCADDR := ADR(data2floor), WRITE := MAIN.write2, TMOUT := t#1s);
fb_floor4ADSwrite(NETID := ads_adr4, PORT := 800, IDXGRP := 16#4020, IDXOFFS := 400, LEN := SIZEOF(data_derevo), SRCADDR := ADR(data_derevo), WRITE := MAIN.write4 OR NOT heartbeat.Q, TMOUT := t#1s);
counter_busy(CU := fb_floor4ADSwrite.BUSY);
counter_error(CU := fb_floor4ADSwrite.ERR);
END_PROGRAM

(* POU HVAC/summer, ST *)
PROGRAM summer
VAR

END_VAR
data1floor[0].3:=heating_mode;

(*--------------------------VITALNYA---------------------------------------------------------------*)

	IF VITALNYA_HVAC.heat_mode=2 THEN (*heat*)
		IF heating_mode THEN VITALNYA_HVAC.zaslinka:=TRUE;(*closed*) ELSE VITALNYA_HVAC.zaslinka:=FALSE; (*opened*)END_IF;
		VITALNYA_HVAC.tepla_pidloga:=TRUE; (*all opened*);
		CASE VITALNYA_HVAC.heat_speed OF
			1:	VITALNYA_HVAC.fancoil_speed:=1;
				IF NOT heating_mode THEN  VITALNYA_HVAC.klapan:=16#0; ELSE VITALNYA_HVAC.klapan:=16#3FFF;END_IF
			2:	VITALNYA_HVAC.fancoil_speed:=2;
				IF NOT heating_mode THEN  VITALNYA_HVAC.klapan:=16#0; ELSE VITALNYA_HVAC.klapan:=16#5FFF;END_IF
			3:	VITALNYA_HVAC.fancoil_speed:=3;
				IF NOT heating_mode THEN  VITALNYA_HVAC.klapan:=16#0; ELSE VITALNYA_HVAC.klapan:=16#7FFF;END_IF
		END_CASE
	END_IF

	IF VITALNYA_HVAC.heat_mode=1 THEN (*cool*)
		IF  heating_mode THEN VITALNYA_HVAC.klapan:=16#0;(*full closed*) END_IF
		IF  heating_mode THEN VITALNYA_HVAC.zaslinka:=FALSE; ELSE VITALNYA_HVAC.zaslinka:=TRUE; END_IF
				VITALNYA_HVAC.tepla_pidloga:=FALSE; (*all closed*)

			CASE VITALNYA_HVAC.heat_speed OF
			1:	VITALNYA_HVAC.fancoil_speed:=1;
				IF NOT heating_mode THEN  VITALNYA_HVAC.klapan:=16#3FFF; ELSE VITALNYA_HVAC.klapan:=16#0;END_IF
			2:	VITALNYA_HVAC.fancoil_speed:=2;
				IF NOT heating_mode THEN  VITALNYA_HVAC.klapan:=16#5FFF; ELSE VITALNYA_HVAC.klapan:=16#0;END_IF
			3:	VITALNYA_HVAC.fancoil_speed:=3;
				IF NOT heating_mode THEN  VITALNYA_HVAC.klapan:=16#7FFF; ELSE VITALNYA_HVAC.klapan:=16#0;END_IF
		END_CASE
	END_IF

	IF VITALNYA_HVAC.heat_mode=3 THEN (*fan*)
		VITALNYA_HVAC.tepla_pidloga:=FALSE;

		CASE VITALNYA_HVAC.heat_speed OF
			1:	VITALNYA_HVAC.fancoil_speed:=0;
				VITALNYA_HVAC.zaslinka:=TRUE;(*closed*)
				VITALNYA_HVAC.klapan:=16#0;(*full closed*)
			2:	VITALNYA_HVAC.fancoil_speed:=2;
				VITALNYA_HVAC.zaslinka:=FALSE;(*opened*)
				VITALNYA_HVAC.klapan:=16#7FFF;
			3:	VITALNYA_HVAC.fancoil_speed:=3;
				VITALNYA_HVAC.zaslinka:=FALSE;(*opened*)
				VITALNYA_HVAC.klapan:=16#7FFF;
		END_CASE
	IF heat.t_out<0 THEN VITALNYA_HVAC.klapan:=16#5FFF; ELSE VITALNYA_HVAC.klapan:=16#0;END_IF
	END_IF



(*--------------------------KABINET---------------------------------------------------------------*)
(*реверс двигуна клапана*)

	IF kabinet_HVAC.heat_mode=2 THEN (*heat*)
		IF heating_mode THEN kabinet_HVAC.zaslinka:=TRUE;(*closed*) ELSE kabinet_HVAC.zaslinka:=FALSE; (*opened*)END_IF;
		kabinet_HVAC.tepla_pidloga:=TRUE; (*all opened*);
		CASE kabinet_HVAC.heat_speed OF
			1:	kabinet_HVAC.fancoil_speed:=1;
				IF heating_mode THEN  kabinet_HVAC.klapan:=16#0; ELSE kabinet_HVAC.klapan:=16#7FFF;END_IF
			2:	kabinet_HVAC.fancoil_speed:=2;
				IF heating_mode THEN  kabinet_HVAC.klapan:=16#0; ELSE kabinet_HVAC.klapan:=16#5FFF;END_IF
			3:	kabinet_HVAC.fancoil_speed:=3;
				IF heating_mode THEN  kabinet_HVAC.klapan:=16#0; ELSE kabinet_HVAC.klapan:=16#3FFF;END_IF
		END_CASE
	END_IF

	IF kabinet_HVAC.heat_mode=1 THEN (*cool*)
		IF NOT heating_mode THEN kabinet_HVAC.klapan:=16#0;(*full closed*) END_IF
		IF NOT heating_mode THEN kabinet_HVAC.zaslinka:=FALSE; ELSE kabinet_HVAC.zaslinka:=TRUE; END_IF
				kabinet_HVAC.tepla_pidloga:=FALSE; (*all closed*)

			CASE kabinet_HVAC.heat_speed OF
			1:	kabinet_HVAC.fancoil_speed:=1;
				IF heating_mode THEN  kabinet_HVAC.klapan:=16#7FFF; ELSE kabinet_HVAC.klapan:=16#0;END_IF
			2:	kabinet_HVAC.fancoil_speed:=2;
				IF heating_mode THEN  kabinet_HVAC.klapan:=16#5FFF; ELSE kabinet_HVAC.klapan:=16#0;END_IF
			3:	kabinet_HVAC.fancoil_speed:=3;
				IF heating_mode THEN  kabinet_HVAC.klapan:=16#3FFF; ELSE kabinet_HVAC.klapan:=16#0;END_IF
		END_CASE
	END_IF

	IF kabinet_HVAC.heat_mode=3 THEN (*fan*)
		kabinet_HVAC.tepla_pidloga:=FALSE;
		IF heat.t_out<0 THEN kabinet_HVAC.klapan:=16#3FFF;(*30%*) ELSE kabinet_HVAC.klapan:=16#0;END_IF
		CASE kabinet_HVAC.heat_speed OF
			1:	kabinet_HVAC.fancoil_speed:=0;
				kabinet_HVAC.zaslinka:=TRUE;(*closed*)
				kabinet_HVAC.klapan:=16#0;(*full closed*)
			2:	kabinet_HVAC.fancoil_speed:=2;
				kabinet_HVAC.zaslinka:=FALSE;(*opened*)
				kabinet_HVAC.klapan:=16#7FFF;
			3:	kabinet_HVAC.fancoil_speed:=3;
				kabinet_HVAC.zaslinka:=FALSE;(*opened*)
				kabinet_HVAC.klapan:=16#7FFF;
		END_CASE
	END_IF


(*--------------------------KINO---------------------------------------------------------------*)
(*реверс двигуна клапана*)

	IF KINO_HVAC.heat_mode=2 THEN (*heat*)
		IF heating_mode THEN KINO_HVAC.zaslinka:=TRUE;(*closed*) ELSE KINO_HVAC.zaslinka:=FALSE; (*opened*)END_IF;
		KINO_HVAC.tepla_pidloga:=TRUE; (*all opened*);
		CASE KINO_HVAC.heat_speed OF
			1:	KINO_HVAC.fancoil_speed:=1;
				IF NOT heating_mode THEN  KINO_HVAC.klapan:=16#0; ELSE KINO_HVAC.klapan:=16#5FFF;END_IF
			2:	KINO_HVAC.fancoil_speed:=2;
				IF NOT heating_mode THEN  KINO_HVAC.klapan:=16#0; ELSE KINO_HVAC.klapan:=16#3FFF;END_IF
			3:	KINO_HVAC.fancoil_speed:=3;
				IF NOT heating_mode THEN  KINO_HVAC.klapan:=16#0; ELSE KINO_HVAC.klapan:=16#0;END_IF
		END_CASE
	END_IF

	IF KINO_HVAC.heat_mode=1 THEN (*cool*)
		IF  heating_mode THEN KINO_HVAC.klapan:=16#7FFF;(*full closed*) END_IF
		IF  heating_mode THEN KINO_HVAC.zaslinka:=FALSE; ELSE KINO_HVAC.zaslinka:=TRUE; END_IF
				KINO_HVAC.tepla_pidloga:=FALSE; (*all closed*)

			CASE KINO_HVAC.heat_speed OF
			1:	KINO_HVAC.fancoil_speed:=1;
				IF NOT heating_mode THEN  KINO_HVAC.klapan:=16#5FFF; ELSE KINO_HVAC.klapan:=16#7FFF;END_IF
			2:	KINO_HVAC.fancoil_speed:=2;
				IF NOT heating_mode THEN  KINO_HVAC.klapan:=16#3FFF; ELSE KINO_HVAC.klapan:=16#7FFF;END_IF
			3:	KINO_HVAC.fancoil_speed:=3;
				IF NOT heating_mode THEN  KINO_HVAC.klapan:=16#0; ELSE KINO_HVAC.klapan:=16#7FFF;END_IF
		END_CASE
	END_IF

	IF KINO_HVAC.heat_mode=3 THEN (*fan*)
		KINO_HVAC.tepla_pidloga:=FALSE;

		CASE KINO_HVAC.heat_speed OF
			1:	KINO_HVAC.fancoil_speed:=0;
				KINO_HVAC.zaslinka:=TRUE;(*closed*)
				KINO_HVAC.klapan:=16#7FFF;(*full closed*)
			2:	KINO_HVAC.fancoil_speed:=2;
				KINO_HVAC.zaslinka:=FALSE;(*opened*)
				KINO_HVAC.klapan:=16#7FFF;
			3:	KINO_HVAC.fancoil_speed:=3;
				KINO_HVAC.zaslinka:=FALSE;(*opened*)
				KINO_HVAC.klapan:=16#7FFF;
		END_CASE
		IF heat.t_out<0 THEN KINO_HVAC.klapan:=16#5FFF;  ELSE KINO_HVAC.klapan:=16#7FFF;END_IF
	END_IF

(*--------------------------DYTJACHA---------------------------------------------------------------*)
(*реверс двигуна клапана*)

	IF dytjacha_HVAC.heat_mode=2 THEN (*heat*)
		IF heating_mode THEN dytjacha_HVAC.zaslinka:=TRUE;(*closed*) ELSE dytjacha_HVAC.zaslinka:=FALSE; (*opened*)END_IF;
		dytjacha_HVAC.tepla_pidloga:=TRUE; (*all opened*);
		CASE dytjacha_HVAC.heat_speed OF
			1:	dytjacha_HVAC.fancoil_speed:=1;
				IF NOT heating_mode THEN  dytjacha_HVAC.klapan:=16#7FFF; ELSE dytjacha_HVAC.klapan:=16#5FFF;END_IF
			2:	dytjacha_HVAC.fancoil_speed:=2;
				IF NOT heating_mode THEN  dytjacha_HVAC.klapan:=16#7FFF; ELSE dytjacha_HVAC.klapan:=16#3FFF;END_IF
			3:	dytjacha_HVAC.fancoil_speed:=3;
				IF NOT heating_mode THEN  dytjacha_HVAC.klapan:=16#7FFF; ELSE dytjacha_HVAC.klapan:=16#0;END_IF
		END_CASE
	END_IF

	IF dytjacha_HVAC.heat_mode=1 THEN (*cool*)
		IF  heating_mode THEN dytjacha_HVAC.klapan:=16#7FFF;(*full closed*) END_IF
		IF  heating_mode THEN dytjacha_HVAC.zaslinka:=FALSE; ELSE dytjacha_HVAC.zaslinka:=TRUE; END_IF
				dytjacha_HVAC.tepla_pidloga:=FALSE; (*all closed*)

			CASE dytjacha_HVAC.heat_speed OF
			1:	dytjacha_HVAC.fancoil_speed:=1;
				IF heating_mode THEN  dytjacha_HVAC.klapan:=16#7FFF; ELSE dytjacha_HVAC.klapan:=16#0;END_IF
			2:	dytjacha_HVAC.fancoil_speed:=2;
				IF heating_mode THEN  dytjacha_HVAC.klapan:=16#5FFF; ELSE dytjacha_HVAC.klapan:=16#0;END_IF
			3:	dytjacha_HVAC.fancoil_speed:=3;
				IF heating_mode THEN  dytjacha_HVAC.klapan:=16#3FFF; ELSE dytjacha_HVAC.klapan:=16#0;END_IF
		END_CASE
	END_IF

	IF dytjacha_HVAC.heat_mode=3 THEN (*fan*)
		dytjacha_HVAC.tepla_pidloga:=FALSE;
		CASE dytjacha_HVAC.heat_speed OF
			1:	dytjacha_HVAC.fancoil_speed:=0;
				dytjacha_HVAC.zaslinka:=TRUE;(*closed*)
				dytjacha_HVAC.klapan:=16#0;(*full closed*)
			2:	dytjacha_HVAC.fancoil_speed:=2;
				dytjacha_HVAC.zaslinka:=FALSE;(*opened*)
				dytjacha_HVAC.klapan:=16#7FFF;
			3:	dytjacha_HVAC.fancoil_speed:=3;
				dytjacha_HVAC.zaslinka:=FALSE;(*opened*)
				dytjacha_HVAC.klapan:=16#7FFF;
		END_CASE
		IF heat.t_out<0 THEN dytjacha_HVAC.klapan:=16#5FFF; ELSE dytjacha_HVAC.klapan:=16#7FFF;END_IF
	END_IF
(*--------------------------SPALNYA---------------------------------------------------------------*)

	IF SPALNYA_HVAC.heat_mode=2 THEN (*heat*)
		IF heating_mode THEN SPALNYA_HVAC.zaslinka:=TRUE;(*closed*) ELSE SPALNYA_HVAC.zaslinka:=FALSE; (*opened*)END_IF;
		SPALNYA_HVAC.tepla_pidloga:=TRUE; (*all opened*);
		CASE SPALNYA_HVAC.heat_speed OF
			1:	SPALNYA_HVAC.fancoil_speed:=1;
				IF NOT  heating_mode THEN  SPALNYA_HVAC.klapan:=16#0; ELSE SPALNYA_HVAC.klapan:=16#3FFF;END_IF
			2:	SPALNYA_HVAC.fancoil_speed:=2;
				IF NOT heating_mode THEN  SPALNYA_HVAC.klapan:=16#0; ELSE SPALNYA_HVAC.klapan:=16#5FFF;END_IF
			3:	SPALNYA_HVAC.fancoil_speed:=3;
				IF NOT heating_mode THEN  SPALNYA_HVAC.klapan:=16#0; ELSE SPALNYA_HVAC.klapan:=16#7FFF;END_IF
		END_CASE
	END_IF

	IF SPALNYA_HVAC.heat_mode=1 THEN (*cool*)
		IF  heating_mode THEN SPALNYA_HVAC.klapan:=16#5FFF;(*full closed*) END_IF
		IF  heating_mode THEN SPALNYA_HVAC.zaslinka:=FALSE; ELSE SPALNYA_HVAC.zaslinka:=TRUE; END_IF
				SPALNYA_HVAC.tepla_pidloga:=FALSE; (*all closed*)

			CASE SPALNYA_HVAC.heat_speed OF
			1:	SPALNYA_HVAC.fancoil_speed:=1;
				IF NOT heating_mode THEN  SPALNYA_HVAC.klapan:=16#3FFF; ELSE SPALNYA_HVAC.klapan:=16#0;END_IF
			2:	SPALNYA_HVAC.fancoil_speed:=2;
				IF NOT heating_mode THEN  SPALNYA_HVAC.klapan:=16#5FFF; ELSE SPALNYA_HVAC.klapan:=16#0;END_IF
			3:	SPALNYA_HVAC.fancoil_speed:=3;
				IF NOT heating_mode THEN  SPALNYA_HVAC.klapan:=16#7FFF; ELSE SPALNYA_HVAC.klapan:=16#0;END_IF
		END_CASE
	END_IF

	IF SPALNYA_HVAC.heat_mode=3 THEN (*fan*)
		SPALNYA_HVAC.tepla_pidloga:=FALSE;
		CASE SPALNYA_HVAC.heat_speed OF
			1:	SPALNYA_HVAC.fancoil_speed:=0;
				SPALNYA_HVAC.zaslinka:=TRUE;(*closed*)
				SPALNYA_HVAC.klapan:=16#0;(*full closed*)
			2:	SPALNYA_HVAC.fancoil_speed:=2;
				SPALNYA_HVAC.zaslinka:=FALSE;(*opened*)
				SPALNYA_HVAC.klapan:=16#0;
			3:	SPALNYA_HVAC.fancoil_speed:=3;
				SPALNYA_HVAC.zaslinka:=FALSE;(*opened*)
				SPALNYA_HVAC.klapan:=16#0;
		END_CASE
		IF heat.t_out<0 THEN SPALNYA_HVAC.klapan:=16#3FFF;(*30%*) ELSE SPALNYA_HVAC.klapan:=16#0;END_IF
	END_IF
END_PROGRAM

(* POU HVAC/winter, ST *)
PROGRAM winter
VAR

END_VAR
(*1-COOL mode 2-HEAT mode, 3-FAN mode*)

(*--------------------------VITALNYA---------------------------------------------------------------*)

	IF VITALNYA_HVAC.heat_mode=2 THEN
				VITALNYA_HVAC.zaslinka:=TRUE;(*closed*)
				VITALNYA_HVAC.tepla_pidloga:=TRUE; (*all opened*)
		CASE VITALNYA_HVAC.heat_speed OF

			1:	VITALNYA_HVAC.fancoil_speed:=1;
				VITALNYA_HVAC.klapan:=16#3FFF;
			2:	VITALNYA_HVAC.fancoil_speed:=2;
				VITALNYA_HVAC.klapan:=16#5FFF;
			3:	VITALNYA_HVAC.fancoil_speed:=3;
				VITALNYA_HVAC.klapan:=16#7FFF;
		END_CASE
	END_IF

	IF VITALNYA_HVAC.heat_mode=1 THEN
				VITALNYA_HVAC.klapan:=16#0;(*full closed*)
				VITALNYA_HVAC.zaslinka:=FALSE;
				VITALNYA_HVAC.tepla_pidloga:=FALSE; (*all closed*)

			CASE VITALNYA_HVAC.heat_speed OF
			1:	VITALNYA_HVAC.fancoil_speed:=1;
			2:	VITALNYA_HVAC.fancoil_speed:=2;
			3:	VITALNYA_HVAC.fancoil_speed:=3;
		END_CASE
	END_IF

	IF VITALNYA_HVAC.heat_mode=3 THEN
		VITALNYA_HVAC.tepla_pidloga:=FALSE;
		IF heat.t_out<0 THEN VITALNYA_HVAC.klapan:=16#3FFF;(*30%*) ELSE VITALNYA_HVAC.klapan:=16#0;END_IF
		CASE VITALNYA_HVAC.heat_speed OF
			1:	VITALNYA_HVAC.fancoil_speed:=0;
				VITALNYA_HVAC.zaslinka:=TRUE;(*closed*)
				VITALNYA_HVAC.klapan:=16#0;(*full closed*)
			2:	VITALNYA_HVAC.fancoil_speed:=2;
				VITALNYA_HVAC.zaslinka:=FALSE;(*opened*)
			3:	VITALNYA_HVAC.fancoil_speed:=3;
				VITALNYA_HVAC.zaslinka:=FALSE;(*opened*)
		END_CASE
	END_IF



(*--------------------------KABINET---------------------------------------------------------------*)
(*реверс двигуна клапана*)

	IF KABINET_HVAC.heat_mode=2 THEN
				KABINET_HVAC.zaslinka:=TRUE;(*closed*)
				KABINET_HVAC.tepla_pidloga:=TRUE; (*all opened*)
		CASE KABINET_HVAC.heat_speed OF

			1:	KABINET_HVAC.fancoil_speed:=1;
				KABINET_HVAC.klapan:=16#5FFF;
			2:	KABINET_HVAC.fancoil_speed:=2;
				KABINET_HVAC.klapan:=16#3FFF;
			3:	KABINET_HVAC.fancoil_speed:=3;
				KABINET_HVAC.klapan:=16#1FFF;
		END_CASE
	END_IF

	IF KABINET_HVAC.heat_mode=1 THEN
				KABINET_HVAC.klapan:=16#7FFF;(*full closed*)
				KABINET_HVAC.zaslinka:=FALSE;
				KABINET_HVAC.tepla_pidloga:=FALSE; (*all closed*)

			CASE KABINET_HVAC.heat_speed OF
			1:	KABINET_HVAC.fancoil_speed:=1;
			2:	KABINET_HVAC.fancoil_speed:=2;
			3:	KABINET_HVAC.fancoil_speed:=3;
		END_CASE
	END_IF

	IF KABINET_HVAC.heat_mode=3 THEN
		KABINET_HVAC.tepla_pidloga:=FALSE;
		IF heat.t_out<0 THEN KABINET_HVAC.klapan:=16#5FFF;(*30%*) ELSE KABINET_HVAC.klapan:=16#7FFF;END_IF
		CASE KABINET_HVAC.heat_speed OF
			1:	KABINET_HVAC.fancoil_speed:=0;
				KABINET_HVAC.zaslinka:=TRUE;(*closed*)
				KABINET_HVAC.klapan:=16#7FFF;(*full closed*)
			2:	KABINET_HVAC.fancoil_speed:=2;
				KABINET_HVAC.zaslinka:=FALSE;(*opened*)
			3:	KABINET_HVAC.fancoil_speed:=3;
				KABINET_HVAC.zaslinka:=FALSE;(*opened*)
		END_CASE
	END_IF



(*--------------------------KINO---------------------------------------------------------------*)
(*реверс двигуна клапана*)
	IF KINO_HVAC.heat_mode=2 THEN
				KINO_HVAC.zaslinka:=TRUE;(*closed*)
				KINO_HVAC.tepla_pidloga:=TRUE; (*all opened*)
		CASE KINO_HVAC.heat_speed OF

			1:	KINO_HVAC.fancoil_speed:=1;
				KINO_HVAC.klapan:=16#5FFF;
			2:	KINO_HVAC.fancoil_speed:=2;
				KINO_HVAC.klapan:=16#3FFF;
			3:	KINO_HVAC.fancoil_speed:=3;
				KINO_HVAC.klapan:=16#1FFF;
		END_CASE
	END_IF

	IF KINO_HVAC.heat_mode=1 THEN
				KINO_HVAC.klapan:=16#0;(*full closed*)
				KINO_HVAC.zaslinka:=FALSE;
				KINO_HVAC.tepla_pidloga:=FALSE; (*all closed*)

			CASE KINO_HVAC.heat_speed OF
			1:	KINO_HVAC.fancoil_speed:=1;
			2:	KINO_HVAC.fancoil_speed:=2;
			3:	KINO_HVAC.fancoil_speed:=3;
		END_CASE
	END_IF

	IF KINO_HVAC.heat_mode=3 THEN
		KINO_HVAC.tepla_pidloga:=FALSE;
		IF heat.t_out<0 THEN KINO_HVAC.klapan:=16#5FFF;(*30%*) ELSE KINO_HVAC.klapan:=16#7FFF;END_IF
		CASE KINO_HVAC.heat_speed OF
			1:	KINO_HVAC.fancoil_speed:=0;
				KINO_HVAC.zaslinka:=TRUE;(*closed*)
				KINO_HVAC.klapan:=16#7FFF;(*full closed*)
			2:	KINO_HVAC.fancoil_speed:=2;
				KINO_HVAC.zaslinka:=FALSE;(*opened*)
			3:	KINO_HVAC.fancoil_speed:=3;
				KINO_HVAC.zaslinka:=FALSE;(*opened*)
		END_CASE
	END_IF



(*--------------------------DYTJACHA---------------------------------------------------------------*)
(*реверс двигуна клапана*)
	IF DYTJACHA_HVAC.heat_mode=2 THEN
				DYTJACHA_HVAC.zaslinka:=TRUE;(*closed*)
				DYTJACHA_HVAC.tepla_pidloga:=TRUE; (*all opened*)
		CASE DYTJACHA_HVAC.heat_speed OF

			1:	DYTJACHA_HVAC.fancoil_speed:=1;
				DYTJACHA_HVAC.klapan:=16#5FFF;
			2:	DYTJACHA_HVAC.fancoil_speed:=2;
				DYTJACHA_HVAC.klapan:=16#3FFF;
			3:	DYTJACHA_HVAC.fancoil_speed:=3;
				DYTJACHA_HVAC.klapan:=16#1FFF;
		END_CASE
	END_IF

	IF DYTJACHA_HVAC.heat_mode=1 THEN
				DYTJACHA_HVAC.klapan:=16#7FFF;(*full closed*)
				DYTJACHA_HVAC.zaslinka:=FALSE;
				DYTJACHA_HVAC.tepla_pidloga:=FALSE; (*all closed*)

			CASE DYTJACHA_HVAC.heat_speed OF
			1:	DYTJACHA_HVAC.fancoil_speed:=1;
			2:	DYTJACHA_HVAC.fancoil_speed:=2;
			3:	DYTJACHA_HVAC.fancoil_speed:=3;
		END_CASE
	END_IF

	IF DYTJACHA_HVAC.heat_mode=3 THEN
		DYTJACHA_HVAC.tepla_pidloga:=FALSE;
		IF heat.t_out<0 THEN DYTJACHA_HVAC.klapan:=16#5FFF;(*30%*) ELSE DYTJACHA_HVAC.klapan:=16#7FFF;END_IF
		CASE DYTJACHA_HVAC.heat_speed OF
			1:	DYTJACHA_HVAC.fancoil_speed:=0;
				DYTJACHA_HVAC.zaslinka:=TRUE;(*closed*)
				DYTJACHA_HVAC.klapan:=16#7FFF;(*full closed*)
			2:	DYTJACHA_HVAC.fancoil_speed:=2;
				DYTJACHA_HVAC.zaslinka:=FALSE;(*opened*)
			3:	DYTJACHA_HVAC.fancoil_speed:=3;
				DYTJACHA_HVAC.zaslinka:=FALSE;(*opened*)
		END_CASE
	END_IF



(*--------------------------SPALNYA---------------------------------------------------------------*)

	IF SPALNYA_HVAC.heat_mode=2 THEN
				SPALNYA_HVAC.zaslinka:=TRUE;(*closed*)
				SPALNYA_HVAC.tepla_pidloga:=TRUE; (*all opened*)
		CASE SPALNYA_HVAC.heat_speed OF

			1:	SPALNYA_HVAC.fancoil_speed:=1;
				SPALNYA_HVAC.klapan:=16#3FFF;
			2:	SPALNYA_HVAC.fancoil_speed:=2;
				SPALNYA_HVAC.klapan:=16#5FFF;
			3:	SPALNYA_HVAC.fancoil_speed:=3;
				SPALNYA_HVAC.klapan:=16#7FFF;
		END_CASE
	END_IF

	IF SPALNYA_HVAC.heat_mode=1 THEN
				SPALNYA_HVAC.klapan:=16#0;(*full closed*)
				SPALNYA_HVAC.zaslinka:=FALSE;
				SPALNYA_HVAC.tepla_pidloga:=FALSE; (*all closed*)

			CASE SPALNYA_HVAC.heat_speed OF
			1:	SPALNYA_HVAC.fancoil_speed:=1;
			2:	SPALNYA_HVAC.fancoil_speed:=2;
			3:	SPALNYA_HVAC.fancoil_speed:=3;
		END_CASE
	END_IF

	IF SPALNYA_HVAC.heat_mode=3 THEN
		SPALNYA_HVAC.tepla_pidloga:=FALSE;
		IF heat.t_out<0 THEN SPALNYA_HVAC.klapan:=16#3FFF;(*30%*) ELSE SPALNYA_HVAC.klapan:=16#0;END_IF
		CASE SPALNYA_HVAC.heat_speed OF
			1:	SPALNYA_HVAC.fancoil_speed:=0;
				SPALNYA_HVAC.zaslinka:=TRUE;(*closed*)
				SPALNYA_HVAC.klapan:=16#0;(*full closed*)
			2:	SPALNYA_HVAC.fancoil_speed:=2;
				SPALNYA_HVAC.zaslinka:=FALSE;(*opened*)
			3:	SPALNYA_HVAC.fancoil_speed:=3;
				SPALNYA_HVAC.zaslinka:=FALSE;(*opened*)
		END_CASE
	END_IF
END_PROGRAM
